# B&R Automation Studio project Soiled_PLC (part 7)

#### 12_sp2Cyclic.ab
```automation-basic
PROGRAM _CYCLIC
	(* cyclic program *)

;---------------------------------------
;Sequence 12 - SP2 Single point 2 D[912]
;---------------------------------------

;Inputs

I_PaddleInPosition		= X[9].X08
I_BagInIncline			= X[9].X07
;I_BagOutAtTop           = X[7].X13

O_OpenBufferStop		= FALSE
O_RunMotor 				= FALSE

I_BagAtOutgoingBuffer	= FALSE
O_OutgoingBufferOpen	= FALSE

Request.IC[1]			= FALSE
Enable.BSF[1]          = FALSE

Alarm[18].Name 			= 0
Alarm[18].Bag			= 10005
Alarm[18].Beacon		= TRUE
Alarm[18].Extra			= 0
Alarm[18].Time			= 3000

;Setup Sequence
STEP = D[918]
;Setup Pulse contact
PLS = (STEP <> LASTSTEP)
LASTSTEP = STEP

;Sequence
;Step 0 - Disabled
IF (STEP = 0) THEN
	;Disabled
ENDIF

;Run Incline until paddle in position
IF (STEP = 1) THEN
	O_RunMotor = NOT I_PaddleInPosition
	IF I_PaddleInPosition THEN
		D[918] = 2
	ENDIF
	IF NOT Std.EStop THEN
		Alarm[18].Name = almSwitchFault
	ENDIF
ENDIF

;request a bag to SP6
IF (STEP = 2) THEN

	IF (Request.BSF[1]  AND NOT Std.HaltSys) THEN
		D[918] = 3
	ENDIF
	;IF (Bag[266].Cat > 0) AND NOT I_BagAtBuffer THEN
		;Alarm[12].Name 	= almBagNotAtProx
		;Alarm[12].Bag	= 266
	;ELSE IF (Bag[266].Cat = 0) AND I_BagAtBuffer THEN
		;Alarm[12].Name 	= almBagNotShownOnScreen
		;Alarm[12].Bag	= 266
	;ENDIF
ENDIF

;Wait for bag to arrive
IF (STEP = 3) THEN
	Enable.BSF[1] 	= TRUE

	IF I_BagInIncline THEN
		D[918] = 4
	ENDIF
	Alarm[18].Name = almBagNotArrived
ENDIF

;Let bag settle at base of incline
TON_10ms((STEP = 4),300,BagSettled,BagSettledET)
IF (STEP = 4) THEN

	IF BagSettled THEN
		D[918] = 5
	ENDIF
ENDIF

;Move Bag up incline
TON_10ms((STEP = 5),500,BagNearTop,BagNearTopET)
TON_10ms(((STEP = 5) AND NOT I_BagInIncline),1000,CloseBufferStop,CloseBufferStopET)
IF (STEP = 5) THEN
	;O_OpenBufferStop 	= NOT CloseBufferStop
	O_RunMotor 			= NOT BagNearTop
	IF BagNearTop  THEN
		D[918] = 6
	ENDIF
	Alarm[18].Name = almSwitchFault
ENDIF

;Check for space at the ongoing buffer
;Run motor for 0.5 seconds
TON_10ms((STEP = 6),50,RunOn,RunOnET)
IF (STEP = 6) THEN
	O_RunMotor 		= NOT RunOn
	IF NOT Std.HaltSys THEN
		Request.IC[1] = TRUE

			IF Enable.IC[1] THEN
				D[918] = 7
			ENDIF

	ENDIF
ENDIF

;Run incline until bag released / arrive at buffer
IF (STEP = 7) THEN
	O_RunMotor 			= TRUE
	;IF PLS THEN
	;	C[13] = 0
	;ENDIF
	IF NOT Enable.IC[1] THEN
		D[918] = 1
	ENDIF
	Alarm[18].Name = almBagNotReleased
ENDIF

;Alarms
TimerAlarm.IN 	= NOT PLS AND (Alarm[18].Name > 0)
TimerAlarm.PT 	= Alarm[18].Time
TimerAlarm FUB TON_10ms()
Alarm[18].On 	= TimerAlarm.Q
Alarm[18].ET 	= TimerAlarm.ET

;Outputs

Y[13].Y04 = O_RunMotor
END_PROGRAM
```

### Program Logical/Sequences/10ms/19_sic_2 (IEC) - * SP2 Empty bags from SDC1/2

#### 12_sp2.var
```iecst
VAR RETAIN
	STEP : UINT;
	PLS : BOOL;
	LASTSTEP : UINT;
END_VAR
VAR
	TimerAlarm : TON_10ms;
	I_BagAtBuffer : BOOL;
	O_OpenBuffer : BOOL;
	SDC2BufferFullET : TIME;
	SDC2BufferFull : BOOL;
	SettledBufferET : TIME;
	SettledBuffer : BOOL;
	O_OpenSP2BufferStop : BOOL;
	O_SelectPoint : BOOL;
	SP2BufferFull : BOOL;
	SP2BufferFullET : UDINT;
	ParingLoopEnabled : BOOL;
	BagInLoopHasDest : BOOL;
	O_OpenSDC1BufferStop : BOOL;
	BagSettledAtBuffer : BOOL;
	BagSettledAtBufferET : UDINT;
	Alternator : USINT;
	I_PaddleInPosition : BOOL;
	I_BagInIncline : BOOL;
	O_OpenBufferStop : BOOL;
	O_RunMotor : BOOL;
	I_BagAtOutgoingBuffer : BOOL;
	O_OutgoingBufferOpen : BOOL;
	BagSettled : BOOL;
	BagSettledET : UDINT;
	BagNearTop : BOOL;
	BagNearTopET : UDINT;
	CloseBufferStop : BOOL;
	CloseBufferStopET : UDINT;
	RunOn : BOOL;
	RunOnET : UDINT;
	I_BagOutAtTop : BOOL;
	BagAtBuffer : BOOL;
	BagAtBufferET : UDINT;
END_VAR
```

#### 12_sp2Cyclic.ab
```automation-basic
PROGRAM _CYCLIC
	(* cyclic program *)

;---------------------------------------
;Sequence 12 - SP2 Single point 2 D[912]
;---------------------------------------

;Inputs

I_BagAtBuffer			= X[9].X09
I_PaddleInPosition		= X[9].X11
I_BagInIncline			= X[9].X10
I_BagOutAtTop           = FALSE ;X[6].X14

O_OpenBufferStop		= FALSE
O_RunMotor 				= FALSE

I_BagAtOutgoingBuffer	= FALSE
O_OutgoingBufferOpen	= FALSE

;Enable.SIC[2]			= FALSE

Alarm[19].Name 			= 0
Alarm[19].Bag			= 10005
Alarm[19].Beacon		= TRUE
Alarm[19].Extra			= 0
Alarm[19].Time			= 3000

;Setup Sequence
STEP = D[919]
;Setup Pulse contact
PLS = (STEP <> LASTSTEP)
LASTSTEP = STEP

;Sequence
;Step 0 - Disabled
IF (STEP = 0) THEN
	;Disabled
ENDIF

;Run Incline until paddle in position
IF (STEP = 1) THEN
	O_RunMotor = NOT I_PaddleInPosition
	IF I_PaddleInPosition THEN
		D[919] = 2
	ENDIF
	IF NOT Std.EStop THEN
		Alarm[19].Name = almSwitchFault
	ENDIF
ENDIF

;Wait for at buffer
TON_10ms(I_BagAtBuffer,300,BagAtBuffer,BagAtBufferET)
IF (STEP = 2) THEN
	IF (BagAtBuffer  AND NOT Std.HaltSys) THEN
		D[919] = 3
	ENDIF
	;IF (Bag[266].Cat > 0) AND NOT I_BagAtBuffer THEN
		;Alarm[12].Name 	= almBagNotAtProx
		;Alarm[12].Bag	= 266
	;ELSE IF (Bag[266].Cat = 0) AND I_BagAtBuffer THEN
		;Alarm[12].Name 	= almBagNotShownOnScreen
		;Alarm[12].Bag	= 266
	;ENDIF
ENDIF

;Open Buffer stop
IF (STEP = 3) THEN
	O_OpenBufferStop 	= TRUE
	;Enable.SIC[1]		= NOT I_BagInIncline
	IF I_BagInIncline THEN
		D[919] = 4
	ENDIF
	Alarm[19].Name = almBagNotArrived
ENDIF

;Let bag settle at base of incline
TON_10ms((STEP = 4),300,BagSettled,BagSettledET)
IF (STEP = 4) THEN
	;O_OpenBufferStop 	= TRUE
	;IF PLS THEN
	;	Bag[265] = Bag[266]
	;	Bag[266] = Bag[0]
	;ENDIF
	IF BagSettled THEN
		D[919] = 5
	ENDIF
ENDIF

;Move Bag up incline
TON_10ms((STEP = 5),500,BagNearTop,BagNearTopET)
TON_10ms(((STEP = 5) AND NOT I_BagInIncline),1000,CloseBufferStop,CloseBufferStopET)
IF (STEP = 5) THEN
	;O_OpenBufferStop 	= NOT CloseBufferStop
	O_RunMotor 			= NOT BagNearTop
	IF BagNearTop THEN
		D[919] = 6
	ENDIF
	Alarm[19].Name = almSwitchFault
ENDIF

;Check for space at the ongoing buffer
;Run motor for 0.5 seconds
TON_10ms((STEP = 6),50,RunOn,RunOnET)
IF (STEP = 6) THEN
	O_RunMotor 		= NOT RunOn
	IF NOT Std.HaltSys THEN
		;IF (Bag[273].Cat = 0) AND NOT I_BagAtOutgoingBuffer AND NOT O_OutgoingBufferOpen THEN
			;IF Line[15].Clear THEN
			IF Line[24].Clear THEN
				D[919] = 7
			;ELSE
			;	Alarm[13].Name = almSwitchFault
			ENDIF
		;ENDIF
	ENDIF
ENDIF

;Run incline until bag released / arrive at buffer
IF (STEP = 7) THEN
	O_RunMotor = TRUE
	IF PLS THEN
		C[24] = 0
	ENDIF
	IF Line[24].Trip THEN
		D[919] = 1
	ENDIF
	Alarm[19].Name = almBagNotReleased
ENDIF

;Alarms
TimerAlarm.IN 	= NOT PLS AND (Alarm[19].Name > 0)
TimerAlarm.PT 	= Alarm[19].Time
TimerAlarm FUB TON_10ms()
Alarm[19].On 	= TimerAlarm.Q
Alarm[19].ET 	= TimerAlarm.ET

;Outputs
Y[9].Y09 = O_OpenBufferStop
Y[13].Y05 = O_RunMotor
END_PROGRAM
```

### Program Logical/Sequences/10ms/8_sl1 (IEC, version 3.00.6) - *Servo Hoist - 3 position

#### sl3.st - Init, cyclic, exit code
```iecst
(********************************************************************
* COPYRIGHT --
********************************************************************
* PROGRAM: sl4.st
* File: sl4.st
* Author: treamsbottom
* Created: March 6 2019
********************************************************************
* Implementation OF PROGRAM Servo Hoist 4 Postion
********************************************************************)
//V2.00.1 First Release
//V2.00.2 FIX - LoadBag wasn;t being set on belt loaded type
//V2.00.3 FIX - 11/08/2019 - Carriage Move alarms were active when the safety zone was off.
//V2.00.4 CHANGE - 11/08/2019 - If the hoist is out of position on loading step- then move to position
//V2.00.5 ADD 12/08/2019 - Add option to stop full bags being bought into service position
//V3.00.1 CHANGE:TR  22/08/2019 - Load Alarms and timer values from config
//V3.00.2 TR 15/09/2019 - Remove EDGEPOS on deviceOut.Bag reference as this doesn;t work with 1_x points as the bag number can change dynamically
//V3.00.3 TR 18/08/2019	- ADD bag check when bag is being loaded.
//V3.00.4 TR 04/10/2019 - FIX: Additional check on Std.MaxCats due to config mode sets to 0 for first scan
//V3.00.5 TR 06/11/2019 - ADD: Alarm when servo hoist is in error.
//V3.00.6 TR 06/11/2019 - FIX: Don;t clear Comm with Comm[0] as unconfiguried tasks can write to Comm[0]
PROGRAM _INIT
//Configuration
mySeq						:= 8;						//Sequence number
MY_VC;						//SET CONSTANT				//Hoist Number Number
myZone 						:= 2;						//Safety Zone
myBag						:= 222;

allowFullBagsInServicePos	:= TRUE;					//Set this to true, if full bags are allowed into service position. Off by default to prevent squashing full bags

//Options
bulkLoaded					:= 0;						//Is the Hoist bulk Loaded.
requestPrgCode				:= 0;						//Request a PRG code from trackview using this d32 register (Start 100 and increase by 20s MAX is 180
CASE Std.PLCStn OF
	0:
		myHoistID				:= 230 + MY_VC;
	1:
		myHoistID				:= 240 + MY_VC;

END_CASE;

//Option to clear the destination when bag arrives,

alarm						ACCESS ADR(Alarm[mySeq]);
bag							ACCESS ADR(Bag[myBag]);
bag_out						ACCESS ADR(Bag[224]);

pHoist 						ACCESS ADR(OpcUa.VC[myHoistID]);
returnStep					ACCESS ADR(D[7970 + MY_VC]);

position_BagOut				:= 1;
position_BagIn				:= 2;
position_Service			:= 3;

i_bagReleased				ACCESS ADR(X[3].X14);
//Outputs
o_safeStopA					ACCESS ADR (Y[0].Y07);
o_safeStopB					ACCESS ADR (Y[0].Y08);
o_guardMoveDown				ACCESS ADR(Hoist_Safety[MY_VC].O_OpenGuard);
o_guardMoveUp				ACCESS ADR(Hoist_Safety[MY_VC].O_CloseGuard);

#if (MY_VC > MAX_HOIST)
	#error 'MAX_HOIST has not been set correctly'
#endif

END_PROGRAM

PROGRAM _CYCLIC

Bag[217].Cat := 1;
Bag[217].Wgt := DINT_TO_UINT(pHoist.Read.Weight/100);
IF (Bag[217].Bid = 0) AND (BidStn > 0) THEN
	Bag[217].Bid := BidStn;
	BidStn := 0;
END_IF;

Request.VC[1]				:= FALSE;

Enable.VC[1]  				:= FALSE;
guardMoveDown				:= FALSE;

//Bit so we can customise the permission to move if required. FOR USE WITH MOVING TOP RAILS
permission_GetBag		:= TRUE;
permission_ReleaseBag	:= TRUE;
permission_Move			:= NOT Std.HaltSysZone[myZone];

pHoist.Write.PermissionToMove := 0;//We have to set permission to move when we want the hoist move.
pHoist.Write.Heartbeat;//This is taken care of in the server task,
pHoist.Write.LoadBag 	:= 0;	//
pHoist.Write.ReceiveBag := 0;	//Cmd to recieve bag
pHoist.Write.ReleaseBag	:= 0;	//Cmd to release bag
pHoist.Write.TargetPosition;	//Set the position of hoist.

autoMode 				:= pHoist.Read.Auto;

IF (myBag = 0) THEN
	alarm.Bag	:= mySeq + 10000;
ELSE
	alarm.Bag	:= myBag;
END_IF;

alarm.Name 		:= 0;
alarm.Beacon	:= TRUE;
alarm.Extra		:= 0;
alarm.Time		:= 3000;

//Setup Sequence
step := D[900 + mySeq];
//Setup Pulse contact
pls := (step <> lastStep);
lastStep := step;

//clear any latched bits
IF pls THEN
	releaseBag := 0;
END_IF;

//Sequence
IF (step = 0) THEN
	//Disabled
END_IF;

//step 1 - move to emptybag in position
IF (step = 1) THEN
	reqPosition := position_BagIn;
	pHoist.Write.PermissionToMove := permission_Move;
	IF (pHoist.Read.PositionNo = reqPosition) AND pHoist.Read.ReadyToReceive THEN
		D[900 + mySeq] := 2;
	END_IF;
	IF autoMode AND permission_Move THEN
		alarm.Name := ALM_CARRIAGE_MOVE_FAULT;
		alarm.Time := 1500;
	END_IF;
END_IF;

//Step 2 - Give permission to recieve bag
IF (step = 2) THEN
	readyToRecieve := ((bag.Cat = 0) AND (pHoist.Read.PositionNo = reqPosition) AND pHoist.Read.ReadyToReceive AND autoMode);
	pHoist.Write.ReceiveBag := 1;
	reqPosition := position_BagIn;
	IF readyToRecieve AND RequestRel.LU[1] THEN // Bag hs been released to empty bag in
		D[900 + mySeq] := 3;
	ELSIF (bag.Cat > 0) THEN
		alarm.Name := ALM_BAG_DATA_ERROR;
	ELSIF (pHoist.Read.PositionNo <> reqPosition) AND autoMode AND permission_Move THEN // Move to position if the buffer hasn;t already been opened.
		pHoist.Write.PermissionToMove := permission_Move;
		alarm.Name := ALM_CARRIAGE_MOVE_FAULT;
		alarm.Time := 1500;
	END_IF;

END_IF;

//Step 3-- Wait for bag to arrive on carriage.
IF (step = 3) THEN
	reqPosition := position_BagIn;
	pHoist.Write.ReceiveBag := 1;
	IF ((bag.Cat = 0) AND (pHoist.Read.PositionNo = reqPosition) AND pHoist.Read.ReadyToReceive AND autoMode AND RequestRel.LU[1]) THEN
		readyToRecieve := 1;
	END_IF;
	Enable.VC[1] := readyToRecieve;
	IF pHoist.Read.ReceiveBag AND (bag.Cat = 0) THEN
		D[900 + mySeq] := 4;
	ELSIF (((pHoist.Read.PositionNo <> reqPosition) OR NOT pHoist.Read.ReadyToReceive ) AND autoMode AND permission_Move) THEN
		alarm.Name := ALM_CARRIAGE_MOVE_FAULT;
		alarm.Time := 1500;
	END_IF;
ELSE
	readyToRecieve := 0;
END_IF;

//step 4 - move to full bag out
IF (step = 4) THEN
	reqPosition := position_BagOut;
	pHoist.Write.PermissionToMove := permission_Move AND permission_ReleaseBag;
	IF (pHoist.Read.PositionNo = reqPosition) AND NOT Enable.PN[1] THEN //We have no feedback for ready to release!! this is checked in the hoist.
		D[900 + mySeq] := step + 1;
	END_IF;
	IF autoMode AND permission_Move  THEN
		alarm.Name := ALM_CARRIAGE_MOVE_FAULT;
		alarm.Time := 1500;
	ELSIF Enable.PN[1] THEN
			alarm.Name := ALM_GENERAL_SEQUENCE;
			alarm.Time := 500;
	END_IF;
	//We should check the hoist status for any alarms??
END_IF;

//step 5 Request Release full bag out
wieghtCheck := (pHoist.Read.Weight < 55000); // hoist sends to 3 decimal places
IF (step = 5) THEN
	okToRelease := Enable.PN[1] AND wieghtCheck AND NOT i_bagReleased;
	reqPosition := position_BagOut;
	requestRelease := (((bag.Cat > 0) OR (myBag = 0) OR Enable.PN[1]) AND (pHoist.Read.PositionNo = reqPosition) AND autoMode AND NOT Std.HaltSysZone[myZone]);
	Request.VC[1]	:= requestRelease;
	IF NOT wieghtCheck THEN
		alarm.Name := almBagOverWeight;
		alarm.Time	:= 500;
	ELSIF requestRelease AND okToRelease  THEN
		D[900 + mySeq] := 6;
	ELSIF (myBag > 0) AND (bag.Cat = 0) THEN
		alarm.Name := ALM_BAG_DATA_ERROR;
		alarm.Time := 0;
	END_IF;
END_IF;

//Step 6 Send the command to release the full bag

bagReleased := (i_bagReleased OR NOT Enable.PN[1]);

IF (step = 6) THEN
	okToRelease :=  Enable.PN[1] AND wieghtCheck;
	reqPosition := position_BagOut;
	IF okToRelease AND (pHoist.Read.PositionNo = reqPosition) AND NOT Std.HaltSysZone[myZone] AND autoMode THEN
		releaseBag := 1;
	END_IF;
	pHoist.Write.ReleaseBag := releaseBag;

	IF NOT wieghtCheck THEN
		alarm.Name := almBagOverWeight;
		alarm.Time	:= 500;
	END_IF;
	IF bagReleased AND releaseBag THEN
//		bag_out := bag;
//		bag := Bag[0];
		D[900 + mySeq] := 1;
	END_IF;
	IF NOT Std.HaltSysZone[myZone] THEN
		alarm.Name := ALM_BAG_NOT_RELEASED;
		alarm.Time := 1500;
	END_IF;
ELSE
	releaseBag := 0;
END_IF;

//Move to service position
IF (step = 90) THEN
	pHoist.Write.PermissionToMove := 1;
	reqPosition := position_Service;
	IF (pHoist.Read.PositionNo = position_Service) THEN //We have no feedback for ready to release!! this is checked in the hoist.
		D[900 + mySeq] := 91;
	END_IF;
	IF autoMode AND permission_Move THEN
		alarm.Name := ALM_CARRIAGE_MOVE_FAULT;
		alarm.Time := 1500;
	END_IF;
END_IF;

//step 91 -- In safe position- Wait for zone to be opened or request to go off
IF (step = 91) THEN
	IF 	SafetyZone[myZone].AccessRequested AND NOT SafetyZone[myZone].Zone_Status THEN
		D[900 + mySeq] := 92;
	ELSIF NOT SafetyZone[myZone].AccessRequested THEN
		D[900 + mySeq] := returnStep;
	ELSIF Hoist_Safety[MY_VC].OutOfPosition THEN
		alarm.Name := ALM_SWITCH_FAULT;
		alarm.Time := 200;
	END_IF;
END_IF;

//step 92 -- Door opened-  wait for safety OK
IF (step = 92) THEN
	IF SafetyZone[myZone].Zone_Status THEN
		D[900 + mySeq] := returnStep;
	END_IF;
END_IF;

IF allowFullBagsInServicePos THEN
	fullBagOnHoist := 0;
ELSE
	fullBagOnHoist := (((bag.Cat > 0) AND (bag.Cat <> Std.MaxCats)) OR ((step > 3) AND (step < 90)));
END_IF;

//Code to request the hoist to move to service position.
IF SafetyZone[myZone].AccessRequested AND (step > 0) AND (step <> 3) AND (step <> 6) AND (step < 90)  AND autoMode AND NOT releaseBag AND NOT fullBagOnHoist THEN
	D[900 + mySeq] := 90;
	CASE step OF
		2:
			returnStep := (step - 1);
		ELSE
			returnStep := step;
	END_CASE;
END_IF;

o_safeStopA	 	:= (step = 3) AND (pHoist.Read.ReadyToReceive OR TestSystem);//Safety stops
o_safeStopB		:= o_safeStopA;

pHoist.Write.BagInTransit := (step = 3) OR releaseBag; //Stop the hoist going into manual mode while a bag is moving.
pHoist.Write.TargetPosition := reqPosition;
o_guardMoveDown := guardMoveDown;
o_guardMoveUp := NOT guardMoveDown;

IF (pHoist.Read.Error OR NOT pHoist.Read.Heartbeat) AND NOT Std.HaltSysZone[myZone] THEN
	alarm.Name := ALM_SERVO_HOIST;
	IF pHoist.Read.Error THEN
		alarm.Time := 400;
	ELSE
		alarm.Time := 3000;
	END_IF;
END_IF;

//Alarms
timerAlarm(IN := NOT pls AND (alarm.Name > 0) AND (alarm.Name = lastAlarm) ,PT:= alarm.Time);
lastAlarm := alarm.Name;

alarm.On 	:= timerAlarm.Q;
alarm.ET 	:= timerAlarm.ET;

END_PROGRAM
```

#### sl3.var - Local variables
```iecst
VAR
	mySeq : UINT;
END_VAR
VAR CONSTANT
	MY_VC : USINT := 1;
END_VAR
VAR
	myZone : USINT;
	myBag : UINT;
	alarm : REFERENCE TO Alm;
	bag : REFERENCE TO Bag_typ;
	bag_out : REFERENCE TO Bag_typ;
	myHoistID : USINT;
	returnStep : REFERENCE TO UINT;
	pHoist : REFERENCE TO OpcUa_VC_type;
	position_BagOut : USINT;
	position_Loading : USINT;
	position_BagIn : USINT;
	position_Service : USINT;
	o_guardMoveUp : REFERENCE TO BOOL;
	o_guardMoveDown : REFERENCE TO BOOL;
	o_safeStopB : REFERENCE TO BOOL;
	o_safeStopA : REFERENCE TO BOOL;
	autoMode : BOOL;
	step : UINT;
	permission_Move : BOOL;
	pls : BOOL;
	lastStep : UINT;
	timerAlarm : TON_10ms;
	reqPosition : USINT;
	readyToRecieve : BOOL;
	okToRelease : BOOL;
	requestRelease : BOOL;
	releaseBag : BOOL;
	f_trig_Released : F_TRIG;
	r_trig_Released : R_TRIG;
	guardMoveDown : BOOL;
	permission_GetBag : BOOL;
	permission_ReleaseBag : BOOL;
	bulkLoaded : BOOL;
	moveGuardDown : BOOL;
	unloadFinished : BOOL;
	myPrg : USINT;
	myCat : UDINT;
	myCus : UDINT;
	myWgt : UINT;
	myMis : UDINT;
	myCnt : UINT;
	myBid : UDINT;
	myDst : UINT;
	myTime : DATE_AND_TIME;
	requestPrgCode : UINT;
	myReportStn : UINT;
	allowFullBagsInServicePos : BOOL; (*Option to allow full bags into service position*)
	fullBagOnHoist : BOOL;
	bagOnCarriage : BOOL;
	lastAlarm : UINT;
	i_bagReleased : REFERENCE TO BOOL;
	bagReleased : BOOL;
	wieghtCheck : BOOL;
END_VAR
```

### Program Logical/Sequences/10ms/10_ebt (IEC) - * EBT Empty bag transfer from SDC2

#### 10_ebt.var
```iecst
VAR RETAIN
	STEP	:UINT;
	PLS	:BOOL;
	LASTSTEP	:UINT;
END_VAR

VAR
	O_OpenBufferStop	:BOOL;
	SettledAtBufferET	:TIME;
	I_BagAtBuffer	:BOOL;
	SettledAtBuffer	:BOOL;
	O_SPI1BufferStopOpen	:BOOL;
	I_BagAtSPI1BufferStop	:BOOL;
	TimerAlarm	:TON_10ms;
	O_SelectPoint	:BOOL;
END_VAR
```

#### 10_ebtCyclic.ab
```automation-basic
PROGRAM _CYCLIC
	(* cyclic program *)

;-----------------------------------------------------
;Sequence 10 - EBT Empty bag transfer from SDC2 D[910]
;-----------------------------------------------------

;Inputs

I_BagAtBuffer			= X[6].X13

O_OpenBufferStop		= FALSE
Enable.DC[1]           = FALSE
O_SelectPoint           = FALSE

I_BagAtSPI1BufferStop	= X[8].X12
O_SPI1BufferStopOpen	= Y[8].Y12

Alarm[10].Name 			= 0
Alarm[10].Bag			= 266
Alarm[10].Beacon		= TRUE
Alarm[10].Extra			= 0
Alarm[10].Time			= 3000

;Setup Sequence
STEP = D[910]
;Setup Pulse contact
PLS = (STEP <> LASTSTEP)
LASTSTEP = STEP

IF (Bag[266].Cat > 0) AND (Bag[266].Bid = 0) AND (BidStn > 0) THEN
	Bag[266].Bid = BidStn
	BidStn = 0
ENDIF

;Sequence
;Step 0 - Disabled
IF (STEP = 0) THEN
	;Disabled
ENDIF

;Step 1 - Wait for space at SPI1 buffer
IF (STEP = 1) THEN
	IF (Line[17].Clear AND NOT I_BagAtSPI1BufferStop AND NOT O_SPI1BufferStopOpen AND NOT Std.HaltSys) THEN
		D[910] = 2
	ENDIF
ENDIF

;Step 2 - Wait for bag at SDC2 empty bag buffer and enable from offgoing
TON_10ms(I_BagAtBuffer,300,SettledAtBuffer,SettledAtBufferET)
IF (STEP = 2) THEN
	IF EnableSDC2Empty THEN
		IF Request.DC[1] THEN
			D[910] = 3
		ELSE IF SettledAtBuffer  THEN
			D[910] = 4
		ENDIF
	ENDIF
ENDIF

;Enable SDC1
IF (STEP = 3) THEN
	Enable.DC[1] = (D[905] <= 2)
	O_SelectPoint = (D[905] <= 2)
	IF PLS THEN
		C[17] = 0
		Bag[266].Prg = Std.MaxProg
		Bag[266].Cat = Std.MaxCats
	ENDIF
	IF Line[17].Trip THEN
		D[910] 		= 1
		Bag[266] 	= Bag[0]
	ENDIF
	Alarm[10].Name = almBagNotArrived
ENDIF

;Step 3 - Transfer empty from SDC2
IF (STEP = 4) THEN
	O_OpenBufferStop = (D[905] <= 2)
	IF PLS THEN
		C[17] = 0
		Bag[266].Prg = Std.MaxProg
		Bag[266].Cat = Std.MaxCats
	ENDIF
	IF Line[17].Trip THEN
		D[910] 		= 1
		Bag[266] 	= Bag[0]
	ENDIF
	Alarm[10].Name = almBagNotArrived
ENDIF

;Alarms
TimerAlarm.IN 	= NOT PLS AND (Alarm[10].Name > 0)
TimerAlarm.PT 	= Alarm[10].Time
TimerAlarm FUB TON_10ms()
Alarm[10].On 	= TimerAlarm.Q
Alarm[10].ET 	= TimerAlarm.ET

;Outputs
Y[6].Y13 = O_OpenBufferStop
Y[8].Y02 = O_SelectPoint
END_PROGRAM
```

### Program Logical/Sequences/10ms/13_spc1 (IEC, version 1.00.0) - * SPC1 Empty bag down

#### 13_spc1Cyclic.ab
```automation-basic
PROGRAM _CYCLIC
	(* cyclic program *)

;----------------------------------------------
;Sequence 13 - SPC1 Pneumatic Conveyor 1 D[913]
;----------------------------------------------

;Inputs
I_CarrAtTop				= X[5].X09
I_CarrAtBottom			= X[5].X10
I_BagOnCarr				= X[5].X11
I_BagReleased			= FALSE ;X[13].X04
I_BagAtBuffer			= X[5].X12

I_BagAtLLBuff			= FALSE ;X[12].X01
O_LLBuffOpen			= FALSE ;Y[12].Y01

O_OpenBuffer			= FALSE
O_MoveCarrUp			= FALSE
O_MoveCarrDown			= FALSE
O_OpenCarrStop			= FALSE

Alarm[13].Name 			= 0
Alarm[13].Bag			= 10013
Alarm[13].Beacon		= FALSE
Alarm[13].Extra			= 0
Alarm[13].Time			= 3000

;Setup Sequence
STEP = D[913]
;Setup Pulse contact
PLS = (STEP <> LASTSTEP)
LASTSTEP = STEP

;Sequence
IF (STEP = 0) THEN
	;Disabled
ENDIF

;Move carriage up to top position
IF (STEP = 1) THEN
	O_MoveCarrUp = TRUE
	IF I_CarrAtTop THEN
		D[913] = 2
	ENDIF
	IF NOT Std.EStop THEN
		Alarm[13].Name = almCarriageMoveFault
	ENDIF
ENDIF

;Check Status
IF (STEP = 2) THEN
	IF (NOT I_BagOnCarr AND NOT I_CarrAtBottom) THEN
		D[913] = 3
	ENDIF
	IF I_BagOnCarr OR I_CarrAtBottom THEN
		Alarm[13].Name = almSwitchFault
	ENDIF
ENDIF

;Wait for bag at buffer
TON_10ms(I_BagAtBuffer,300,SettledBuffer,SettledBufferET)
IF (STEP = 3) THEN
	IF SettledBuffer AND NOT Std.HaltSys THEN
		D[913] = 4
	ENDIF
ENDIF

;Open Buffer stop - Enable
IF (STEP = 4) THEN
	O_OpenBuffer 	= (NOT I_BagOnCarr AND I_CarrAtTop)
	;Enable.SVC[4] 	= (NOT I_BagOnCarr AND I_CarrAtBottom)
	IF I_BagOnCarr THEN
		D[913] = 5
	ENDIF
	Alarm[13].Name = almBagNotArrived
ENDIF

;Let bag settle on carriage
TON_10ms(I_BagOnCarr,300,BagSettledOnCarr,BagSettledOnCarrET)
IF (STEP = 5) THEN
	IF BagSettledOnCarr THEN
		D[913] = 6
	ENDIF
	Alarm[13].Name = almBagNotSettled
ENDIF

;Move Carriage down to bottom position
IF (STEP = 6) THEN
	O_MoveCarrDown = TRUE
	IF I_CarrAtBottom THEN
		D[913] = 7
	ENDIF
	IF NOT Std.EStop THEN
		Alarm[13].Name = almCarriageMoveFault
	ENDIF
ENDIF

;Check if buffer is clear
IF (STEP = 7) THEN
	;IF (Line[33].Clear AND NOT I_BagAtLLBuff AND NOT O_LLBuffOpen AND NOT Std.HaltSysLoading) THEN
	IF Enable.BSN[1] THEN
		D[913] = 8
	ENDIF
	;IF NOT Std.HaltSys THEN
	;	IF I_BagReleased THEN
	;		Alarm[13].Name = almSwitchFault
	;	ENDIF
	;ENDIF
ENDIF

;Open carriage stop let bag into buffer
IF (STEP = 8) THEN
	O_OpenCarrStop = TRUE
	;IF PLS THEN
	;	C[33] = 0
	;ENDIF
	;IF Line[33].Trip THEN
	IF NOT Enable.BSN[1] THEN
		D[913] = 9
	ENDIF
	IF NOT Std.EStop THEN
		Alarm[13].Name = almBagNotReleased
	ENDIF
ENDIF

;Check Top position switch
IF (STEP = 9) THEN
	IF NOT I_CarrAtTop THEN
		D[913] = 1
	ENDIF
	Alarm[13].Name = almSwitchFault
ENDIF

;Alarms
TimerAlarm.IN 	= NOT PLS AND (Alarm[13].Name > 0)
TimerAlarm.PT 	= Alarm[13].Time
TimerAlarm FUB TON_10ms()
Alarm[13].On 	= TimerAlarm.Q
Alarm[13].ET 	= TimerAlarm.ET

;PLC Outputs
;-----------
Y[7].Y16 		= (O_OpenBuffer 	AND I_CarrAtTop)
Y[2].Y03 		= (O_MoveCarrUp 	AND NOT I_CarrAtTop)
Y[2].Y07 		= (O_MoveCarrDown 	AND NOT I_CarrAtBottom)
Y[2].Y12 		= (O_OpenCarrStop 	AND I_CarrAtBottom)

;Don't allow forcing of carriage movement and carriage stop
YForceDisable[7].Y16 = TRUE
YForceDisable[2].Y03 = TRUE
YForceDisable[2].Y07 = TRUE
YForceDisable[2].Y12 = TRUE

END_PROGRAM
```

#### 13_spc1.var
```iecst
VAR RETAIN
	I_CarrAtTop	:BOOL;
	I_CarrAtBottom	:BOOL;
	STEP	:UINT;
	PLS	:BOOL;
	LASTSTEP	:UINT;
	O_MoveCarrUp	:BOOL;
	O_OpenCarrStop	:BOOL;
	O_MoveCarrDown	:BOOL;
	I_BagOnCarr	:BOOL;
END_VAR

VAR
	O_OpenBuffer	:BOOL;
	SettledBuffer	:BOOL;
	SettledBufferET	:TIME;
	I_BagAtBuffer	:BOOL;
	BagSettledOnCarr	:BOOL;
	BagSettledOnCarrET	:TIME;
	I_BagReleased	:BOOL;
	TimerAlarm	:TON_10ms;
	I_BagAtLLBuff	:BOOL;
	O_LLBuffOpen	:BOOL;
END_VAR
```

### Program Logical/Sequences/10ms/16_sdc3 (IEC, version 1.00.0) - * SDC3 Wash-extractors

#### 16_sdc3Cyclic.ab
```automation-basic
PROGRAM _CYCLIC
	(* cyclic program *)

;Sequence 16 - Discharger 3 D[916]

;-----------------------------------------
;Revision 1.00 19/12/2005 D.J. First Issue
;-----------------------------------------

DischargerEnable 		= (NOT Std.HaltSys)

I_BagAtBuffer			= FALSE
I_BagAtDischarger		= X[8].X07
I_OpenBag				= X[8].X08
I_LoadDropped			= X[8].X08
I_BagReleased			= FALSE
I_BagEmpty			  	= TRUE

I_BagAtEmptyBuffer		= FALSE ;X[11].X07
O_EmptyBagBufferOpen	= FALSE ;Y[11].Y07

O_BagReady				= FALSE
O_OpenBuffer 			= FALSE
O_Steadys				= FALSE
O_Closer				= FALSE
O_OpenBag				= FALSE
O_OpenStop				= FALSE

;Enable.DC[1]			= FALSE
Request.DC[3]			= FALSE

;Alarm
Alarm[16].Name 			= almNoAlarm ;Clear sequence alarm name
Alarm[16].Bag 			= 263
Alarm[16].Beacon		= TRUE
Alarm[16].Extra			= 0
Alarm[16].Time			= 3000

;Setup Sequence
STEP = D[916]
;Setup Pulse contact
PLS = (STEP <> LASTSTEP)
LASTSTEP = STEP

;Step 0 - Disabled
IF (STEP = 0) THEN
	;Disabled
ENDIF

;Check Status - Bag settled at buffer, no bag at discharger, bag at buffer on screen and no bag at discharger on the screen
TON_10ms(I_BagAtBuffer,300,SettledAtBuffer,SettledAtBufferET)
IF (STEP = 1) THEN
	;IF (DischargerEnable AND SettledAtBuffer AND NOT I_BagAtDischarger AND (Bag[261].Cat > 0) AND (Bag[263].Cat = 0) AND NOT Std.HaltSys) THEN
	IF (DischargerEnable AND NOT I_BagAtDischarger AND (Bag[263].Cat = 0) AND NOT Std.HaltSys) THEN
		D[916] = 2
	ENDIF
	IF (Bag[263].Cat > 0) THEN
		Alarm[16].Name = almBagDataError
	ELSE IF I_BagAtDischarger THEN
		Alarm[16].Name = almSwitchFault
	;ELSE IF (Bag[263].Cat > 0) AND NOT I_BagAtBuffer THEN
	;	Alarm[16].Name 	= almBagDataError
	;	Alarm[16].Bag	= 263
	;ELSE IF (Bag[261].Cat = 0) AND I_BagAtBuffer THEN
	;	Alarm[16].Name 	= almBagNotShownOnScreen
	;	Alarm[16].Bag	= 261
	ENDIF
ENDIF

;Wait for bag in discharger
IF (STEP = 2) THEN
	;Enable.DC[1]	= TRUE
	;O_OpenBuffer 	= TRUE
	IF I_BagAtDischarger THEN
		D[916] = 3
	ENDIF
	;Alarm[16].Name = almBagNotArrived
ENDIF

;Let bag settle in discharger
TON_10ms(((STEP = 3) AND I_BagAtDischarger),1000,SettledAtDischarger,SettledAtDischargerET)
IF (STEP = 3) THEN
	IF PLS  AND (Bag[263].Cat = 0) AND (Bag[252].Cat > 0) THEN
		Bag[252].Dst = 0
		Bag[263]     = Bag[252]
		Bag[252]     = Bag[0]
	ENDIF
	IF SettledAtDischarger THEN
		D[916] = 4
	ENDIF
	IF (Bag[263].Cat = Std.MaxCats) THEN
		D[916] = 11
	ENDIF
	Alarm[16].Name = almBagNotSettled
ENDIF

;Allow steadys to move down
TON_10ms((STEP = 4),400,SteadysDown,SteadysDownET)
IF (STEP = 4) THEN
	IF (SteadysDown AND NOT I_OpenBag) THEN
		D[916] = 5
	ENDIF
	IF I_OpenBag THEN
		Alarm[16].Name = almSwitchFault
	ENDIF
ENDIF

;Steady cylinders on from steps 4 - 9
O_Steadys = ((STEP >= 4) AND (STEP <= 9))

;Bag opener on from step 5 - 8
O_OpenBag = ((STEP >= 6) AND (STEP <= 8))

;Bag Ready to Washing Machine
IF (STEP = 5) THEN
	O_BagReady = TRUE
	IF I_OpenBag OR TestDischarger THEN
		D[916] = 6
	ENDIF
ENDIF

;Set LoadDropped to False
IF (STEP <> 6) THEN
	LoadDropped = FALSE
ENDIF

;Open Bag Until LoadDropped recieved and has been open for 6 seconds
TON_10ms((STEP = 6),600,MinOpen,MinOpenET) ;ET means Elapsed Time
IF (STEP = 6) THEN

	IF NOT I_OpenBag OR TestDischarger THEN
	;IF I_BagEmpty THEN
		LoadDropped = TRUE
	ENDIF

	IF (LoadDropped AND MinOpen) THEN
		;Write Report
		;------------
		IF (ReportUnloading[3].Cat = 0) THEN
			ReportUnloading[3].Cat = UINT(Bag[263].Cat)	;Category
			ReportUnloading[3].Cus = Bag[263].Cus		;Customer
			ReportUnloading[3].Wgt = Bag[263].Wgt		;Weight
			ReportUnloading[3].Cnt = 0					;Count
			ReportUnloading[3].Stn = 0					;Station
			ReportUnloading[3].Mcn = 3					;Machine
		ENDIF
	ENDIF
	IF (LoadDropped AND MinOpen) THEN
		D[916] = 7
	ENDIF
	Alarm[16].Name = almLoadNotDropped
ENDIF

;Change display to empty bag
IF (STEP = 7) THEN
	O_BagReady = Std.Clock500ms
	IF (I_OpenBag OR TestDrop) THEN
		Bag[263].Prg 	= Std.MaxProg
		Bag[263].Cat 	= Std.MaxCats
		D[916] 			= 8
	ENDIF
	Alarm[16].Name = almGeneralSequence
ENDIF

;Close bag
TON_10ms((STEP = 8),700,CloserDown,CloserDownET)
IF (STEP = 8) THEN
	O_Closer = TRUE
	IF CloserDown THEN
		D[916] = 9
	ENDIF
ENDIF

;Allow closer to go back up
TON_10ms((STEP = 9),700,CloserUp,CloserUpET)
IF (STEP = 9) THEN
	IF CloserUp THEN
		D[916] = 10
	ENDIF
ENDIF

;Allow steadys to go up
TON_10ms((STEP = 10),400,SteadyUp,SteadyUpET)
IF (STEP = 10) THEN
	IF SteadyUp THEN
		D[916] = 11
	ENDIF
ENDIF

;Check for space on empty bag buffer
IF (STEP = 11) THEN
	Request.DC[3] = TRUE
	IF Enable.DC[3] THEN
		D[916] = 12
	ENDIF
ENDIF

;Open buffer stop - unitl bag out
IF (STEP = 12) THEN
	O_OpenStop 	= TRUE
	Bag[263] 	= Bag[0]
	IF NOT Enable.DC[3] THEN
		D[916] = 1
	ENDIF
	Alarm[16].Name = almBagNotReleased
ENDIF

;Alarms
TimerAlarm.IN 	= NOT PLS AND (Alarm[16].Name > 0)
TimerAlarm.PT 	= Alarm[16].Time
TimerAlarm FUB TON_10ms()
Alarm[16].On 	= TimerAlarm.Q
Alarm[16].ET 	= TimerAlarm.ET

;Outputs
Y[8].Y08 	= O_BagReady
;Y[6].Y01 	= O_OpenBuffer
Y[8].Y09 	= O_Steadys
Y[8].Y10 	= O_OpenBag
Y[8].Y05 	= O_Closer
Y[8].Y11 	= O_OpenStop
END_PROGRAM
```

#### 16_sdc3.var
```iecst
VAR RETAIN
	STEP	:UINT;
	PLS	:BOOL;
	LASTSTEP	:UINT;
	SteadyUp	:BOOL;
	CloserUpET	:TIME;
	SteadysDown	:BOOL;
	SteadysDownET	:TIME;
	LoadDropped	:BOOL;
	SteadyUpET	:TIME;
	CloserDownET	:TIME;
	SettledAtDischargerET	:TIME;
	MinOpenET	:TIME;
	SettledAtDischarger	:BOOL;
	CloserDown	:BOOL;
	MinOpen	:BOOL;
	CloserUp	:BOOL;
	SettledAtBuffer	:BOOL;
	SettledAtBufferET	:TIME;
	I_BagAtBuffer	:BOOL;
	O_OpenStop	:BOOL;
	O_OpenBag	:BOOL;
	O_Steadys	:BOOL;
	O_OpenBuffer	:BOOL;
	O_Closer	:BOOL;
	I_BagAtDischarger	:BOOL;
	I_OpenBag	:BOOL;
	I_LoadDropped	:BOOL;
	TestDrop	:BOOL;
END_VAR

VAR
	DischargerEnable	:BOOL;
	TestDischarger	:BOOL;
	I_BagEmpty	:BOOL;
	O_BagReady	:BOOL;
	I_BagReleased	:BOOL;
	O_EmptyBagBufferOpen	:BOOL;
	I_BagAtEmptyBuffer	:BOOL;
	TimerAlarm	:TON_10ms;
	CodeStep	:BOOL;
	BCD_BIN_CAT	:BCD_BIN_OUTPUT;
	BCD_BIN_CUS	:BCD_BIN_OUTPUT;
	BCD_BIN_WGT	:BCD_BIN_OUTPUT;
END_VAR
```

### Program Logical/Sequences/10ms/19_sic2 (IEC) - *incline

#### ic.st
```iecst
(********************************************************************
 * COPYRIGHT --
 ********************************************************************
 * Program: ic
 * File: ic.st
 * Author: treamsbottom
 * Created: July 17, 2015
 ********************************************************************
 * Implementation of program Incline conveyor.
 ********************************************************************)
//V1.00.1 First Release
PROGRAM _INIT
//Configuration
mySeq					:= 19;		//Sequence number
myIO					:= 10; 	//Incline Conveyor IO module number
myIC					:= 2;		//Incline Conveyor Number
useRequest				:= FALSE; 	//Use the Request bit. Only use when working with x_1_point. otherwise use RequestRelease as the i_bagAtBuffer.
myBuffBag				:= 261;		//Ingoing Buffer bag number
myBag					:= 259;		//Incline bag number
myRelLine				:= 32;
myOutBag				:= Line[myRelLine].LastBag;	//Outgoing buffer bag number

myZone 					:= 0;
//Timer Values
bufferSettleTime		:= 300;  	// Time for bag to settle at buffer in.
moveUpInclineTime		:= 8;//>>IN SECONDS<< // Time to move bag up incline after closing stop.//Min of 4 to shut buffer stop....

alarm						ACCESS ADR(Alarm[mySeq]);
bag							ACCESS ADR(Bag[myBag]);
bag_buff					ACCESS ADR(Bag[myBuffBag]);
bag_out						ACCESS ADR(Bag[myOutBag]);
line_release				ACCESS ADR(Line[myRelLine]);
END_PROGRAM

PROGRAM _CYCLIC
//Inputs
i_paddleInPosition		:= X[myIO].X03;
i_bagAtBuffer			:= X[myIO].X01;
i_bagInIncline			:= X[myIO].X02;
i_BagReleased			:= FALSE;//X[myIO].X05;  //<--- Bag release trip- only to be used in special cases. Take when using tracked bags, as the next sequence will need to copy data into a transit position

i_bagAtBufferOut 		:= X[11].X03; // Any Single bag buffer out IO.
i_bufferOutOpen			:= Y[11].Y03;

//End of inputs.

o_openBuffer			:= FALSE;
o_runMotor				:= FALSE;

Request.IC[myIC] 		:= FALSE;
RequestRel.IC[myIC] 	:= FALSE;

IF (myBag = 0) THEN
	alarm.Bag	:= mySeq + 10000;
ELSE
	alarm.Bag	:= myBag;
END_IF;

alarm.Name 		:= 0;
alarm.Beacon		:= TRUE;
alarm.Extra		:= 0;
alarm.Time		:= 3000;

//Setup Sequence
step := D[900 + mySeq];
//Setup Pulse contact
pls := (step <> laststep);
laststep := step;

//Sequence
IF (step = 0) THEN
	//Disabled
END_IF;

//Run Incline until paddle in position
IF (step = 1) THEN
	o_runMotor := NOT i_paddleInPosition;
	IF i_paddleInPosition THEN
		D[900 + mySeq] := 2;
		Count[mySeq] := Count[mySeq] + 1;
	END_IF;
	IF NOT Std.HaltSysZone[myZone] THEN
		alarm.Name := ALM_SWITCH_FAULT;
	END_IF;
END_IF;

//Wait for at buffer
ton_10ms_SettledBuffer(IN:= i_bagAtBuffer, PT:= bufferSettleTime);
IF (step = 2) THEN
	IF NOT i_bagInIncline THEN
		IF useRequest THEN
			D[900 + mySeq] := 3;
		ELSE
			IF ton_10ms_SettledBuffer.Q THEN
				IF (myBuffBag > 0) THEN
					IF (bag_buff.Cat > 0) AND (bag.Cat = 0) THEN
						D[900 + mySeq] := 3;
					ELSIF (bag_buff.Cat = 0) THEN
						alarm.Name := ALM_BAG_DATA_ERROR;
						alarm.Bag := myBuffBag;
					ELSE
						alarm.Name := ALM_BAG_DATA_ERROR;
					END_IF;
				ELSE
					D[900 + mySeq] := 3;
				END_IF;
			ELSIF (myBuffBag > 0) AND (bag_buff.Cat > 0) THEN
				alarm.Name := ALM_BAG_NOT_SETTLED;
			END_IF;
		END_IF;
	ELSE
		alarm.Name := ALM_SWITCH_FAULT;
	END_IF;
END_IF;

//Open Buffer stop
IF (step = 3) THEN
	releaseValid := ((myBag = 0) OR ((bag.Cat = 0) AND (bag_buff.Cat > 0)));
	o_openBuffer	   := releaseValid AND NOT useRequest;
	Request.IC[myIC]  := releaseValid AND useRequest;
	IF i_bagInIncline AND releaseValid THEN
		IF (myBag > 0) THEN
			bag := bag_buff; //Clear empty buffer bag data if used
			bag_buff := Bag[0];
		END_IF;
		D[900 + mySeq] := 4;
	ELSIF (myBag > 0) THEN
		IF (bag.Cat > 0) THEN
			alarm.Name := ALM_BAG_DATA_ERROR;
			alarm.Time := 0;
		ELSIF (bag_buff.Cat = 0) THEN
			alarm.Name := ALM_BAG_DATA_ERROR;
			alarm.Bag := myBuffBag;
			alarm.Time := 0;
		ELSE
			alarm.Name  := ALM_BAG_NOT_ARRIVED;
		END_IF;
	ELSE
		alarm.Name  := ALM_BAG_NOT_ARRIVED;
	END_IF;
END_IF;

ton_10ms_SettledIncline(IN:= (step = 4), PT:= 300);
IF (step = 4) THEN
	o_openBuffer := NOT useRequest;
	IF ton_10ms_SettledIncline.Q THEN
		D[900 + mySeq] := 5;
	END_IF;
END_IF;

//Move Bag up incline
ctu_moveUpIncline(CU:=(step = 5) AND NOT Std.HaltSysZone[myZone] AND Std.Clock1s, RESET := (step <> 5), PV := moveUpInclineTime);
IF (step = 5) THEN
	o_openBuffer 	:= (ctu_moveUpIncline.CV <= 4) AND NOT useRequest;//Close buffer stop after 3 seconds running..
	o_runMotor 		:= TRUE;
	IF ctu_moveUpIncline.Q THEN
		D[900 + mySeq] := 6;
	ELSIF NOT Std.HaltSysZone[myZone] THEN
		alarm.Name := ALM_SWITCH_FAULT;
	END_IF;

END_IF;

//Check for line space.
IF (step = 6) THEN
	releaseValid := (NOT i_bagAtBufferOut AND NOT i_bufferOutOpen AND NOT i_BagReleased AND ((myBag = 0) OR ((bag.Cat > 0) AND (bag_out.Cat = 0))));
	IF (myRelLine > 0) THEN
		IF (line_release.Clear AND releaseValid) THEN
			C[myRelLine] := 0;
			D[900 + mySeq] := 7;
		END_IF;
		IF (line_release.Clear AND i_bagAtBufferOut) THEN
			alarm.Name := ALM_SWITCH_FAULT;
		ELSIF (myBag > 0) AND (bag.Cat = 0) THEN
			alarm.Name := ALM_BAG_DATA_ERROR;
			alarm.Time := 0;
		ELSIF line_release.Clear AND (myOutBag > 0) AND (bag_out.Cat > 0) THEN
			alarm.Name := ALM_BAG_DATA_ERROR;
			alarm.Bag := myOutBag;
			alarm.Time := 0;
		END_IF;
	ELSE
		RequestRel.IC[myIC] := releaseValid;
		IF EnableRel.IC[myIC] AND releaseValid THEN

			D[900 + mySeq] := 7;
		ELSIF (myBag > 0) AND (bag.Cat = 0) THEN
			alarm.Name := ALM_BAG_DATA_ERROR;
			alarm.Time := 0;
		ELSIF (myOutBag > 0) AND (bag_out.Cat > 0) THEN
			alarm.Name := ALM_BAG_DATA_ERROR;
			alarm.Bag := myOutBag;
			alarm.Time := 0;
		END_IF;
	END_IF;
	IF i_BagReleased THEN
		alarm.Name := ALM_SWITCH_FAULT;
		alarm.Time := 0;
	END_IF;
	releaseValid := 0; //Clear this as we are using it as a latch in line 7
END_IF;

//Run motor to release bag.
IF (step = 7) THEN
	IF (NOT i_bagAtBufferOut AND NOT i_bufferOutOpen AND ((myBag = 0) OR ((bag.Cat > 0) AND (bag_out.Cat = 0)))) THEN
		releaseValid := 1;
	END_IF;
	o_runMotor := releaseValid AND NOT Std.HaltSysZone[myZone];
	IF releaseValid THEN
		IF (myBag = 0) THEN
			IF (myRelLine > 0) THEN
				IF line_release.Trip THEN
					D[900 + mySeq] := 1;
				END_IF;
			ELSE
				IF NOT EnableRel.IC[myIC] OR i_BagReleased THEN
					D[900 + mySeq] := 1;
				END_IF;
			END_IF;
			IF NOT Std.HaltSysZone[myZone] THEN
				alarm.Name := ALM_BAG_NOT_RELEASED;
			END_IF;
		ELSE//Use tracking
			IF (myRelLine > 0) THEN
				IF line_release.Trip THEN
					bag_out := bag;
					bag := Bag[0];
					D[900 + mySeq] := 1;
				END_IF;
			ELSE
				IF (i_BagReleased OR NOT EnableRel.IC[myIC]) AND (bag.Cat = 0)  THEN // Make sure data is copied out by enabling sequence.
					D[900 + mySeq] := 1;
				ELSIF NOT EnableRel.IC[myIC] AND (bag.Cat > 0) THEN
					alarm.Name := ALM_BAG_DATA_ERROR;
				END_IF;
			END_IF;
		END_IF;
	ELSIF i_bagAtBufferOut OR i_bufferOutOpen THEN
			alarm.Name := ALM_SWITCH_FAULT;
			alarm.Time := 0;
	ELSIF (myBag > 0) THEN
		IF (bag.Cat = 0) THEN
			alarm.Name := ALM_BAG_DATA_ERROR;
			alarm.Time := 0;
		ELSIF (bag_out.Cat > 0) THEN
			alarm.Name := ALM_BAG_DATA_ERROR;
			alarm.Bag := myOutBag;
			alarm.Time := 0;
		END_IF;
	END_IF;
END_IF;

//-----------------------------------
//PLC Outputs - adjust TO suit system
//-----------------------------------

Y[2].Y14	:= o_runMotor;
Y[myIO].Y01 := o_openBuffer;

//Alarms
timerAlarm(IN := NOT pls AND (alarm.Name > 0),PT:= alarm.Time);

alarm.On 	:= timerAlarm.Q;
alarm.ET 	:= timerAlarm.ET;;

END_PROGRAM
```

### Program Logical/Sequences/10ms/27_sic1 (IEC, version 1.00.5) - *incline

#### ic.st - Implementation code
```iecst
(********************************************************************
 * COPYRIGHT --
 ********************************************************************
 * Program: ic
 * File: ic.st
 * Author: treamsbottom
 * Created: July 17, 2015
 ********************************************************************
 * Implementation of program Incline conveyor.
 ********************************************************************)
//V1.00.1 First Release
PROGRAM _INIT
//Configuration
mySeq					:= 9;		//Sequence number
myIO					:= 6; 	//Incline Conveyor IO module number
myIC					:= 1;		//Incline Conveyor Number
useRequest				:= FALSE; 	//Use the Request bit. Only use when working with x_1_point. otherwise use RequestRelease as the i_bagAtBuffer.
myBuffBag				:= 240;		//Ingoing Buffer bag number
myBag					:= 241;		//Incline bag number
myRelLine				:= 0;
myOutBag				:= Line[myRelLine].LastBag;	//Outgoing buffer bag number

myZone 					:= 0;
//Timer Values
bufferSettleTime		:= 300;  	// Time for bag to settle at buffer in.
moveUpInclineTime		:= 8;//>>IN SECONDS<< // Time to move bag up incline after closing stop.//Min of 4 to shut buffer stop....

alarm						ACCESS ADR(Alarm[mySeq]);
bag							ACCESS ADR(Bag[myBag]);
bag_buff					ACCESS ADR(Bag[myBuffBag]);
bag_out						ACCESS ADR(Bag[myOutBag]);
line_release				ACCESS ADR(Line[myRelLine]);
END_PROGRAM

PROGRAM _CYCLIC
//Inputs
i_paddleInPosition		:= X[myIO].X15;
i_bagAtBuffer			:= X[8].X06;
i_bagInIncline			:= X[myIO].X14;
i_BagReleased			:= FALSE;//X[myIO].X05;  //<--- Bag release trip- only to be used in special cases. Take when using tracked bags, as the next sequence will need to copy data into a transit position

i_bagAtBufferOut 		:= FALSE; // Any Single bag buffer out IO.
i_bufferOutOpen			:= FALSE;

//End of inputs.

o_openBuffer			:= FALSE;
o_runMotor				:= FALSE;

Request.IC[myIC] 		:= FALSE;
RequestRel.IC[myIC] 	:= FALSE;

IF (myBag = 0) THEN
	alarm.Bag	:= mySeq + 10000;
ELSE
	alarm.Bag	:= myBag;
END_IF;

alarm.Name 		:= 0;
alarm.Beacon		:= TRUE;
alarm.Extra		:= 0;
alarm.Time		:= 3000;

//Setup Sequence
step := D[900 + mySeq];
//Setup Pulse contact
pls := (step <> laststep);
laststep := step;

//Sequence
IF (step = 0) THEN
	//Disabled
END_IF;

//Run Incline until paddle in position
IF (step = 1) THEN
	o_runMotor := NOT i_paddleInPosition;
	IF i_paddleInPosition THEN
		D[900 + mySeq] := 2;
		Count[mySeq] := Count[mySeq] + 1;
	END_IF;
	IF NOT Std.HaltSysZone[myZone] THEN
		alarm.Name := ALM_SWITCH_FAULT;
	END_IF;
END_IF;

//Wait for at buffer
ton_10ms_SettledBuffer(IN:= i_bagAtBuffer, PT:= bufferSettleTime);
IF (step = 2) THEN
	IF NOT i_bagInIncline THEN
		IF useRequest THEN
			D[900 + mySeq] := 3;
		ELSE
			IF ton_10ms_SettledBuffer.Q THEN
				IF (myBuffBag > 0) THEN
					IF (bag_buff.Cat > 0) AND (bag.Cat = 0) THEN
						D[900 + mySeq] := 3;
					ELSIF (bag_buff.Cat = 0) THEN
						alarm.Name := ALM_BAG_DATA_ERROR;
						alarm.Bag := myBuffBag;
					ELSE
						alarm.Name := ALM_BAG_DATA_ERROR;
					END_IF;
				ELSE
					D[900 + mySeq] := 3;
				END_IF;
			ELSIF (myBuffBag > 0) AND (bag_buff.Cat > 0) THEN
				alarm.Name := ALM_BAG_NOT_SETTLED;
			END_IF;
		END_IF;
	ELSE
		alarm.Name := ALM_SWITCH_FAULT;
	END_IF;
END_IF;

//Open Buffer stop
IF (step = 3) THEN
	releaseValid := ((myBag = 0) OR ((bag.Cat = 0) AND (bag_buff.Cat > 0)));
	o_openBuffer	   := releaseValid AND NOT useRequest;
	Request.IC[myIC]  := releaseValid AND useRequest;
	IF i_bagInIncline AND releaseValid THEN
		IF (myBag > 0) THEN
			bag := bag_buff; //Clear empty buffer bag data if used
			bag_buff := Bag[0];
		END_IF;
		D[900 + mySeq] := 4;
	ELSIF (myBag > 0) THEN
		IF (bag.Cat > 0) THEN
			alarm.Name := ALM_BAG_DATA_ERROR;
			alarm.Time := 0;
		ELSIF (bag_buff.Cat = 0) THEN
			alarm.Name := ALM_BAG_DATA_ERROR;
			alarm.Bag := myBuffBag;
			alarm.Time := 0;
		ELSE
			alarm.Name  := ALM_BAG_NOT_ARRIVED;
		END_IF;
	ELSE
		alarm.Name  := ALM_BAG_NOT_ARRIVED;
	END_IF;
END_IF;

ton_10ms_SettledIncline(IN:= (step = 4), PT:= 300);
IF (step = 4) THEN
	o_openBuffer := NOT useRequest;
	IF ton_10ms_SettledIncline.Q THEN
		D[900 + mySeq] := 5;
	END_IF;
END_IF;

//Move Bag up incline
ctu_moveUpIncline(CU:=(step = 5) AND NOT Std.HaltSysZone[myZone] AND Std.Clock1s, RESET := (step <> 5), PV := moveUpInclineTime);
IF (step = 5) THEN
	o_openBuffer 	:= (ctu_moveUpIncline.CV <= 4) AND NOT useRequest;//Close buffer stop after 3 seconds running..
	o_runMotor 		:= TRUE;
	IF ctu_moveUpIncline.Q THEN
		D[900 + mySeq] := 6;
	ELSIF NOT Std.HaltSysZone[myZone] THEN
		alarm.Name := ALM_SWITCH_FAULT;
	END_IF;

END_IF;

//Check for line space.
IF (step = 6) THEN
	releaseValid := (NOT i_bagAtBufferOut AND NOT i_bufferOutOpen AND NOT i_BagReleased AND ((myBag = 0) OR ((bag.Cat > 0) AND (bag_out.Cat = 0))));
	IF (myRelLine > 0) THEN
		IF (line_release.Clear AND releaseValid) THEN
			C[myRelLine] := 0;
			D[900 + mySeq] := 7;
		END_IF;
		IF (line_release.Clear AND i_bagAtBufferOut) THEN
			alarm.Name := ALM_SWITCH_FAULT;
		ELSIF (myBag > 0) AND (bag.Cat = 0) THEN
			alarm.Name := ALM_BAG_DATA_ERROR;
			alarm.Time := 0;
		ELSIF line_release.Clear AND (myOutBag > 0) AND (bag_out.Cat > 0) THEN
			alarm.Name := ALM_BAG_DATA_ERROR;
			alarm.Bag := myOutBag;
			alarm.Time := 0;
		END_IF;
	ELSE
		RequestRel.IC[myIC] := releaseValid;
		IF EnableRel.IC[myIC] AND releaseValid THEN

			D[900 + mySeq] := 7;
		ELSIF (myBag > 0) AND (bag.Cat = 0) THEN
			alarm.Name := ALM_BAG_DATA_ERROR;
			alarm.Time := 0;
		ELSIF (myOutBag > 0) AND (bag_out.Cat > 0) THEN
			alarm.Name := ALM_BAG_DATA_ERROR;
			alarm.Bag := myOutBag;
			alarm.Time := 0;
		END_IF;
	END_IF;
	IF i_BagReleased THEN
		alarm.Name := ALM_SWITCH_FAULT;
		alarm.Time := 0;
	END_IF;
	releaseValid := 0; //Clear this as we are using it as a latch in line 7
END_IF;

//Run motor to release bag.
IF (step = 7) THEN
	IF (NOT i_bagAtBufferOut AND NOT i_bufferOutOpen AND ((myBag = 0) OR ((bag.Cat > 0) AND (bag_out.Cat = 0)))) THEN
		releaseValid := 1;
	END_IF;
	o_runMotor := releaseValid AND NOT Std.HaltSysZone[myZone];
	IF releaseValid THEN
		IF (myBag = 0) THEN
			IF (myRelLine > 0) THEN
				IF line_release.Trip THEN
					D[900 + mySeq] := 1;
				END_IF;
			ELSE
				IF NOT EnableRel.IC[myIC] OR i_BagReleased THEN
					D[900 + mySeq] := 1;
				END_IF;
			END_IF;
			IF NOT Std.HaltSysZone[myZone] THEN
				alarm.Name := ALM_BAG_NOT_RELEASED;
				alarm.Time := 6000;
			END_IF;
		ELSE//Use tracking
			IF (myRelLine > 0) THEN
				IF line_release.Trip THEN
					bag_out := bag;
					bag := Bag[0];
					D[900 + mySeq] := 1;
				END_IF;
			ELSE
				IF (i_BagReleased OR NOT EnableRel.IC[myIC]) AND (bag.Cat = 0)  THEN // Make sure data is copied out by enabling sequence.
					D[900 + mySeq] := 1;
				ELSIF NOT EnableRel.IC[myIC] AND (bag.Cat > 0) THEN
					alarm.Name := ALM_BAG_DATA_ERROR;
				END_IF;
			END_IF;
		END_IF;
	ELSIF i_bagAtBufferOut OR i_bufferOutOpen THEN
			alarm.Name := ALM_SWITCH_FAULT;
			alarm.Time := 0;
	ELSIF (myBag > 0) THEN
		IF (bag.Cat = 0) THEN
			alarm.Name := ALM_BAG_DATA_ERROR;
			alarm.Time := 0;
		ELSIF (bag_out.Cat > 0) THEN
			alarm.Name := ALM_BAG_DATA_ERROR;
			alarm.Bag := myOutBag;
			alarm.Time := 0;
		END_IF;
	END_IF;
END_IF;

//-----------------------------------
//PLC Outputs - adjust TO suit system
//-----------------------------------

Y[2].Y09	:= o_runMotor;
Y[8].Y06	:= o_openBuffer;

//Alarms
timerAlarm(IN := NOT pls AND (alarm.Name > 0),PT:= alarm.Time);

alarm.On 	:= timerAlarm.Q;
alarm.ET 	:= timerAlarm.ET;;

END_PROGRAM
```

### Program Logical/Sequences/10ms/21_sbsn_1 (IEC) - * SP2 Empty bags from SDC1/2

#### 12_sp2.var
```iecst
VAR RETAIN
	STEP : UINT;
	PLS : BOOL;
	LASTSTEP : UINT;
END_VAR
VAR
	TimerAlarm : TON_10ms;
	I_BagAtBuffer : BOOL;
	O_OpenBuffer : BOOL;
	SDC2BufferFullET : TIME;
	SDC2BufferFull : BOOL;
	SettledBufferET : TIME;
	SettledBuffer : BOOL;
	O_OpenSP2BufferStop : BOOL;
	O_SelectPoint : BOOL;
	SP2BufferFull : BOOL;
	SP2BufferFullET : UDINT;
	ParingLoopEnabled : BOOL;
	BagInLoopHasDest : BOOL;
	O_OpenSDC1BufferStop : BOOL;
	BagSettledAtBuffer : BOOL;
	BagSettledAtBufferET : UDINT;
	Alternator : USINT;
	I_PaddleInPosition : BOOL;
	I_BagInIncline : BOOL;
	O_OpenBufferStop : BOOL;
	O_RunMotor : BOOL;
	I_BagAtOutgoingBuffer : BOOL;
	O_OutgoingBufferOpen : BOOL;
	BagSettled : BOOL;
	BagSettledET : UDINT;
	BagNearTop : BOOL;
	BagNearTopET : UDINT;
	CloseBufferStop : BOOL;
	CloseBufferStopET : UDINT;
	RunOn : BOOL;
	RunOnET : UDINT;
	I_BagOutAtTop : BOOL;
	BagAtBuffer : BOOL;
	BagAtBufferET : UDINT;
	I_BagStackerNearFull : BOOL;
	BagStackerHasSpace : BOOL;
	BagStackerHasSpaceET : UDINT;
	SIC3BufferFull : BOOL;
	SIC3BufferFullET : UDINT;
	I_OnLineA : BOOL;
	I_TiltA : BOOL;
	I_TiltB : BOOL;
	I_Bagout : BOOL;
	O_SelectLineA : BOOL;
	O_SelectLineB : BOOL;
	O_OpenStops : BOOL;
	O_TiltCylinder : BOOL;
	O_OperatePusher : BOOL;
	PointReset : BOOL;
	PointResetET : UDINT;
	BagAtTilt : BOOL;
	BagAtTiltET : UDINT;
	TiltDown : BOOL;
	TiltDownET : UDINT;
	TiltUp : BOOL;
	TiltUpET : UDINT;
	NotFull : BOOL;
	NotFullET : UDINT;
	Pushed : BOOL;
	SBSN1 : BOOL;
	SBSN1ET : UDINT;
	RequirePusherET : UDINT;
	PushedET : UDINT;
	Pusher : BOOL;
	PusherET : UDINT;
	O_Pusher : BOOL;
END_VAR
```

#### 12_sp2Cyclic.ab
```automation-basic
PROGRAM _CYCLIC
	(* cyclic program *)

;---------------------------------------
;Sequence 12 - SP2 Single point 2 D[912]
;---------------------------------------

;Inputs

I_OnLineA		  		= X[7].X01
I_TiltA					= X[7].X02
I_TiltB					= X[7].X03
I_Bagout				= X[7].X04

O_OpenBufferStop		= FALSE
O_SelectLineA			= FALSE
O_SelectLineB			= FALSE
O_OpenStops				= FALSE
O_TiltCylinder			= FALSE
O_OperatePusher			= FALSE
O_Pusher                = FALSE

Request.BSN[1]			= FALSE
Enable.SP[5]            = FALSE

Alarm[21].Name 			= 0
Alarm[21].Bag			= 10010
Alarm[21].Beacon		= TRUE
Alarm[21].Extra			= 0
Alarm[21].Time			= 3000

;Setup Sequence
STEP = D[921]
;Setup Pulse contact
PLS = (STEP <> LASTSTEP)
LASTSTEP = STEP

;Sequence
IF (STEP = 0) THEN
	;Disabled
ENDIF

;Select Line 'A'
TON_10ms((STEP = 1),100,PointReset,PointResetET)
IF (STEP = 1) THEN
	O_SelectLineA = NOT PointReset
	IF PointReset AND NOT Std.HaltSys THEN
		D[921] = 2
	ENDIF
ENDIF

;give request to SP5
IF ((STEP = 2) OR (STEP = 3)) THEN
	Request.BSN[1] = TRUE
ENDIF

;give request to SP5
;TON_10ms(I_BagAtBuffer,300,BagAtBuffer,BagAtBufferET)
IF (STEP = 2) THEN

	IF Enable.BSN[1] THEN
		D[921] = 3
	ENDIF
ENDIF

;Open buffer stop
IF (STEP = 3) THEN
	O_SelectLineA 		= TRUE
	;O_OpenBufferStop 	= TRUE
	;Enable.SP[5]		= NOT I_OnLineA
	IF I_OnLineA THEN
		D[921] = 4
	ENDIF
	Alarm[21].Name = almBagNotArrived
ENDIF

;Select Line 'B' and Wait for bag in Tilt position
TON_10ms((I_TiltA AND I_TiltB),300,BagAtTilt,BagAtTiltET)
IF (STEP = 4) THEN
	O_SelectLineB = TRUE
	IF BagAtTilt THEN
		D[921] = 5
	ENDIF
	Alarm[21].Name = almBagNotSettled
ENDIF

;Tilt down
TON_10ms((STEP = 5),500,TiltDown,TiltDownET)
TON_10ms(TiltDown,300,Pusher,PusherET)
IF (STEP = 5) THEN
	O_TiltCylinder = TRUE
	O_Pusher       = TiltDown
	IF Pusher THEN
		D[921] = 6
	ENDIF
ENDIF

;Tilt up
TON_10ms((STEP = 6),500,TiltUp,TiltUpET)
IF (STEP = 6) THEN
	IF TiltUp THEN
		D[921] = 7
	ENDIF
	Alarm[21].Time			= 1000
	Alarm[21].Name = almDestinationNotValid
ENDIF

;Check not full
TON_10ms(NOT I_Bagout,300,NotFull,NotFullET)
IF (STEP = 7) THEN
	IF NotFull THEN
		D[921] = 8
	ENDIF
	Alarm[21].Name = almBagNotReleased
ENDIF

;Open stops to release bag
IF (STEP = 8) THEN
	O_OpenStops = TRUE
	IF I_Bagout THEN
		D[921] = 1
	ENDIF
	Alarm[21].Name = almBagNotReleased
ENDIF

;Pusher Cylinder
TON_10ms(I_Bagout AND NOT Pushed,200,SBSN1,SBSN1ET)
TON_10ms((STEP = 8)  AND NOT Pushed,500,O_OperatePusher,RequirePusherET)
TON_10ms(O_OperatePusher,500,Pushed,PushedET)

;ton_10ms_o_operatePusher(IN:= (step = 8) AND NOT ton_10ms_Pushed.Q, PT:= 500);
;ton_10ms_Pushed(IN:= o_operatePusher, PT:= 500);

;Alarms
TimerAlarm.IN 	= NOT PLS AND (Alarm[21].Name > 0)
TimerAlarm.PT 	= Alarm[21].Time
TimerAlarm FUB TON_10ms()
Alarm[21].On 	= TimerAlarm.Q
Alarm[21].ET 	= TimerAlarm.ET

;Outputs
;Y[7].Y01 = O_OpenBufferStop
Y[7].Y01 = O_SelectLineA
Y[7].Y02 = O_SelectLineB
Y[7].Y04 = O_TiltCylinder
Y[7].Y05 = O_OpenStops
Y[7].Y03 = O_OperatePusher
Y[7].Y14 = O_Pusher
END_PROGRAM
```

### Program Logical/Sequences/10ms/22_sbsf_1 (IEC) - * SP2 Empty bags from SDC1/2

#### 12_sp2.var
```iecst
VAR RETAIN
	STEP : UINT;
	PLS : BOOL;
	LASTSTEP : UINT;
END_VAR
VAR
	TimerAlarm : TON_10ms;
	I_BagAtBuffer : BOOL;
	O_OpenBuffer : BOOL;
	SDC2BufferFullET : TIME;
	SDC2BufferFull : BOOL;
	SettledBufferET : TIME;
	SettledBuffer : BOOL;
	O_OpenSP2BufferStop : BOOL;
	O_SelectPoint : BOOL;
	SP2BufferFull : BOOL;
	SP2BufferFullET : UDINT;
	ParingLoopEnabled : BOOL;
	BagInLoopHasDest : BOOL;
	O_OpenSDC1BufferStop : BOOL;
	BagSettledAtBuffer : BOOL;
	BagSettledAtBufferET : UDINT;
	Alternator : USINT;
	I_PaddleInPosition : BOOL;
	I_BagInIncline : BOOL;
	O_OpenBufferStop : BOOL;
	O_RunMotor : BOOL;
	I_BagAtOutgoingBuffer : BOOL;
	O_OutgoingBufferOpen : BOOL;
	BagSettled : BOOL;
	BagSettledET : UDINT;
	BagNearTop : BOOL;
	BagNearTopET : UDINT;
	CloseBufferStop : BOOL;
	CloseBufferStopET : UDINT;
	RunOn : BOOL;
	RunOnET : UDINT;
	I_BagOutAtTop : BOOL;
	BagAtBuffer : BOOL;
	BagAtBufferET : UDINT;
	I_BagStackerNearFull : BOOL;
	BagStackerHasSpace : BOOL;
	BagStackerHasSpaceET : UDINT;
	SIC3BufferFull : BOOL;
	SIC3BufferFullET : UDINT;
	I_OnLineA : BOOL;
	I_TiltA : BOOL;
	I_TiltB : BOOL;
	I_Bagout : BOOL;
	O_SelectLineA : BOOL;
	O_SelectLineB : BOOL;
	O_OpenStops : BOOL;
	O_TiltCylinder : BOOL;
	O_OperatePusher : BOOL;
	PointReset : BOOL;
	PointResetET : UDINT;
	BagAtTilt : BOOL;
	BagAtTiltET : UDINT;
	TiltDown : BOOL;
	TiltDownET : UDINT;
	TiltUp : BOOL;
	TiltUpET : UDINT;
	NotFull : BOOL;
	NotFullET : UDINT;
	Pushed : BOOL;
	SBSN1 : BOOL;
	SBSN1ET : UDINT;
	RequirePusherET : UDINT;
	PushedET : UDINT;
	I_RockSepA : BOOL;
	I_RockSepB : BOOL;
	I_OutLineA : BOOL;
	I_OutLineB : BOOL;
	O_OpenRockSep : BOOL;
	O_LevelCylinder : BOOL;
	O_OpenLineAStop : BOOL;
	O_OpenLineBStop : BOOL;
	LevelClear : BOOL;
	LevelClearET : UDINT;
	SettledInSeps : BOOL;
	SettledInSepsET : UDINT;
	SettledLevel : BOOL;
	SettledLevelET : UDINT;
	LevellerDown : BOOL;
	LevellerDownET : UDINT;
	LevellerUp : BOOL;
	LevellerUpET : UDINT;
	O_LevelCylinderUP : BOOL;
	PRLineClearET : ARRAY[0..5] OF UDINT;
END_VAR
```

#### 12_sp2Cyclic.ab
```automation-basic
PROGRAM _CYCLIC
	(* cyclic program *)

;---------------------------------------
;Sequence 12 - SP2 Single point 2 D[912]
;---------------------------------------

;Inputs
I_RockSepA				= X[7].X07
I_RockSepB				= X[7].X08
I_TiltA					= X[7].X09
I_TiltB					= X[7].X10
I_OutLineA				= X[7].X06
I_OutLineB				= X[7].X11

O_OpenRockSep			= FALSE
O_LevelCylinder			= FALSE
O_OpenLineAStop			= FALSE
O_OpenLineBStop			= FALSE
O_SelectLineA			= FALSE
O_SelectLineB			= FALSE

Request.BSF[1]         = FALSE

Alarm[22].Name 			= 0
Alarm[22].Bag			= 10011
Alarm[22].Beacon		= TRUE
Alarm[22].Extra			= 0
Alarm[22].Time			= 3000

;Setup Sequecne
STEP = D[922]
;Setup Pulse contact
PLS = (STEP <> LASTSTEP)
LASTSTEP = STEP

;Sequence

;Select Line 'A'
TON_10ms((NOT I_TiltA AND NOT I_TiltB),100,LevelClear,LevelClearET)
IF (STEP = 1) THEN
	IF LevelClear AND NOT Std.HaltSys THEN
		D[922] = 2
	ENDIF
	Alarm[22].Name = almSwitchFault
ENDIF

;Open seperators wait for leveller to be ready
TON_10ms(((STEP = 2) AND I_RockSepA AND I_RockSepB),200,SettledInSeps,SettledInSepsET)
IF (STEP = 2) THEN
	O_OpenRockSep = TRUE
	IF SettledInSeps THEN
		D[922] = 3
	ENDIF
	;Alarm[22].Name = almBagNotArrived
ENDIF

;Wait for bag to settle in leveller position
TON_10ms((I_TiltA AND I_TiltB),300,SettledLevel,SettledLevelET)
IF (STEP = 3) THEN
	IF SettledLevel THEN
		D[922] = 4
	ENDIF
	Alarm[22].Name = almBagNotSettled
ENDIF

;Move bag leveller down
TON_10ms((STEP = 4),500,LevellerDown,LevellerDownET)
IF (STEP = 4) THEN
	O_LevelCylinder = TRUE
	IF LevellerDown THEN
		D[922] = 5
	ENDIF
ENDIF

;Allow bag leveller to retract
TON_10ms((STEP = 5),500,LevellerUp,LevellerUpET)
IF (STEP = 5) THEN
	O_LevelCylinderUP = TRUE
	IF LevellerUp THEN
		D[922] = 6
	ENDIF
ENDIF

;Check room in Buffer
IF (STEP = 6) THEN
	IF NOT Std.HaltSys THEN
		Request.BSF[1] = TRUE
		IF Enable.BSF[1] THEN
			D[922] = 7
		ENDIF
	ENDIF
ENDIF

O_SelectLineA = ((STEP <> 8) AND (STEP <> 9))

;Open stop on line 'A'
IF (STEP = 7) THEN
	O_OpenLineAStop = TRUE
	;IF PLS THEN
	;	C[17] = 0
	;ENDIF
	IF I_OutLineA THEN
		D[922] = 8
	ENDIF
	Alarm[22].Name = almBagNotReleased
ENDIF

;Open stop on line 'B'
IF (STEP = 8) THEN
	O_OpenLineBStop = TRUE
	IF I_OutLineB THEN
		D[922] = 9
	ENDIF
	Alarm[22].Name = almBagNotReleased
ENDIF

;Select bag stop and wait for bag out of leveller
IF (STEP = 9) THEN
	O_SelectLineB = TRUE
	IF NOT Enable.BSF[1] THEN
		D[922] = 1
	ENDIF
	Alarm[22].Name = almBagNotReleased
ENDIF

;Alarms
TimerAlarm.IN 	= NOT PLS AND (Alarm[22].Name > 0)
TimerAlarm.PT 	= Alarm[22].Time
TimerAlarm FUB TON_10ms()
Alarm[22].On 	= TimerAlarm.Q
Alarm[22].ET 	= TimerAlarm.ET

;Outputs
Y[7].Y08 = O_OpenRockSep
Y[7].Y11 = O_LevelCylinder
Y[7].Y09 = O_OpenLineAStop
Y[7].Y10 = O_OpenLineBStop
Y[7].Y07 = O_SelectLineA
Y[7].Y06 = O_SelectLineB

;SBS Offgoing Bagstacker Pressure relief
TON_10ms((NOT X[7].X12 AND NOT X[7].X13),500,Y[7].Y12,PRLineClearET[0])

;SPR1-3
TON_10ms((NOT X[4].X13 AND NOT X[4].X14),500,Y[4].Y13,PRLineClearET[1])
TON_10ms((NOT X[5].X13 AND NOT X[5].X14),500,Y[5].Y13,PRLineClearET[2])
TON_10ms((NOT X[4].X13 AND NOT X[7].X14),500,Y[7].Y14,PRLineClearET[3])
TON_10ms((NOT X[7].X15 AND NOT X[7].X16),500,Y[7].Y15,PRLineClearET[4])
END_PROGRAM
```

### Program Logical/Sequences/10ms/24_slu_2 (IEC) - * Loading unit SLU1

#### 3_slu_1.var
```iecst
VAR RETAIN
	STEP : UINT;
	PLS : BOOL;
	LASTSTEP : UINT;
	EBagSettled : BOOL;
	EBagSettledET : TIME;
	O_OpenStop : BOOL;
	O_SteadyCylinders : BOOL;
	LoadingUnitClear : BOOL;
	LoadingUnitClearET : TIME;
END_VAR
VAR
	CompressCount : UINT;
	O_MoveCompressorUp : BOOL;
	SteadysUpET : TIME;
	SteadysUp : BOOL;
	SteadysDown : BOOL;
	SteadysDownET : TIME;
	I_BagAtBuffer : BOOL;
	O_OpenBufferStop : BOOL;
	I_BagInLoadingUnit : BOOL;
	I_BagFrontPast : BOOL;
	SwitchFault : BOOL;
	TimerAlarm : TON_10ms;
	I_CompressorAtTop : BOOL;
	I_CompressorAtBot : BOOL;
	I_CompressorAtMid : BOOL;
	O_MoveCompressorDn : BOOL;
	BagSettledBuffer : BOOL;
	BagSettledBufferET : TIME;
	I_BagAtSVC1Buffer : BOOL;
	O_SVC1BufferOpen : BOOL;
	I_ChuteBlocked : BOOL;
	CompressorDn : BOOL;
	CompressorDnET : UDINT;
	O_MoveDownTop : BOOL;
	O_MoveDownBottom : BOOL;
	CompressorUp : BOOL;
	CompressorUpET : UDINT;
	O_ElephantsFoot : BOOL;
	HaltDownStairs : BOOL;
	I_BagAtSIC1Buffer : BOOL;
	O_SIC1BufferOpen : BOOL;
	BagDropped : BOOL;
	ChuteClear : BOOL;
	ChuteClearET : UDINT;
END_VAR
```

#### 3_slu_1Cyclic.ab
```automation-basic
PROGRAM _CYCLIC
	(* cyclic program *)

;--------------------------------
;Sequence 3 - Loading Unit D[903]
;--------------------------------

;Inputs / Ouputs

I_BagAtBuffer			= X[11].X11
I_BagFrontPast			= X[8].X12
I_BagInLoadingUnit		= X[8].X11

I_ChuteBlocked			= X[8].X16
HaltDownStairs          = NOT X[6].X12

;O_MoveCompressorUp		= FALSE
Request.LU[2]  		= FALSE

I_BagAtSIC1Buffer		= X[11].X15 ;X[12].X11
O_SIC1BufferOpen		= Y[11].Y15 ;Y[12].Y11

O_OpenBufferStop		= FALSE
O_SteadyCylinders		= FALSE
O_OpenStop	 			= FALSE

Enable.SDP[1]			= FALSE

Alarm[24].Name 			= 0
Alarm[24].Bag			= 287
Alarm[24].Beacon		= TRUE
Alarm[24].Extra			= 0
Alarm[24].Time			= 3000

;Setup Sequence
;--------------
STEP = D[924]
;Setup Pulse contact
PLS = (STEP <> LASTSTEP)
LASTSTEP = STEP

IF (STEP = 0) THEN
	;Disabled
ENDIF

;Wait for Empty bag at buffer
SwitchFault = (I_BagFrontPast OR I_BagInLoadingUnit)
TON_10ms(NOT SwitchFault,200,LoadingUnitClear,LoadingUnitClearET)
TON_10ms(I_BagAtBuffer,300,BagSettledBuffer,BagSettledBufferET)
IF (STEP = 1) THEN
	IF BagSettledBuffer AND LoadingUnitClear AND NOT HaltDownStairs THEN
	;IF LoadingUnitClear AND NOT Std.HaltSys THEN
		D[924] = 2
	ENDIF
	IF SwitchFault THEN
		Alarm[24].Name = almSwitchFault
	ENDIF
ENDIF

;Open stops let bag in Loading Unit
IF (STEP = 2) THEN
	O_OpenStop 			= TRUE
	O_OpenBufferStop 	= TRUE
	;Enable.SLU[1]		= NOT I_BagFrontPast
	IF I_BagFrontPast THEN
		D[924] = 3
	ENDIF
	Alarm[24].Name = almBagNotArrived
ENDIF

;Wait for bag to settle
TON_10ms(I_BagInLoadingUnit,700,EBagSettled,EBagSettledET)
IF (STEP = 3) THEN
	IF EBagSettled THEN
		D[924] = 4
	ENDIF
	Alarm[23].Name = almBagNotSettled
ENDIF

;Steady cylinders on from steps 4 - 5
O_SteadyCylinders = ((STEP >= 4) AND (STEP <= 8))

;Move Steady Cylinders down
TON_10ms((STEP = 4),300,SteadysDown,SteadysDownET)
IF (STEP = 4) THEN
	IF (SteadysDown AND (Bag[287].Cat = 0)) THEN
		D[924] = 5
	ENDIF
	IF (Bag[287].Cat <> 0) THEN
		Alarm[4].Name = almBagDataError
	ELSE
		Alarm[4].Name = almNoAlarm
	ENDIF
ENDIF

IF ((NOT STEP = 6) AND (NOT STEP = 8)) THEN
	BagDropped = FALSE
ENDIF

;Wait for request from spd 1
IF (STEP = 5) THEN

	IF Request.SDP[1] THEN
		D[924] = 6
	ENDIF
ENDIF

IF (NOT (STEP = 6) AND NOT (STEP = 8)) THEN
	BagDropped = FALSE
ENDIF

;Wait for linen to pass photo cell
TON_10ms(NOT I_ChuteBlocked,300,ChuteClear,ChuteClearET)
IF (STEP = 6) THEN
	Enable.SDP[1] = TRUE
	Request.LU[2] = TRUE

	IF I_ChuteBlocked THEN
		BagDropped = TRUE
	ENDIF
	IF BagDropped AND ChuteClear and (Bag[287].Cat > 0)and (Bag[287].Wgt < 649)THEN
		D[924] = 9
	ELSE IF BagDropped AND ChuteClear and (Bag[287].Cat > 0)and (Bag[287].Wgt > 649)THEN
		D[924] = 9
	ENDIF

ENDIF

;Wait for request from SDP1
IF (STEP = 7) THEN
	IF (Request.SDP[1] AND (Bag[285].Cat = Bag[287].Cat) AND (Bag[287].Wgt < 650)) THEN
		IF Request.SDP[1] THEN
			D[924] = 8
		ENDIF
	ELSE IF (Request.SDP[1] AND (Bag[285].Cat <> Bag[287].Cat)) THEN
		D[924] = 9
	ELSE IF (Bag[287].Wgt > 650)THEN
		D[924] = 9
	ENDIF
ENDIF

;Wait for linen to pass photo cell
TON_10ms((STEP = 6),300,SteadysUp,SteadysUpET)
IF (STEP = 8) THEN
	Enable.SDP[1] = TRUE
	Request.LU[2] = TRUE
	IF I_ChuteBlocked THEN
		BagDropped = TRUE
	ENDIF
	IF BagDropped AND ChuteClear THEN
		D[924] = 9
	ENDIF
ENDIF

;Allow Steady Cylinders to move up
TON_10ms((STEP = 9),300,SteadysUp,SteadysUpET)
IF (STEP = 9) THEN
	IF SteadysUp THEN
		D[924] = 10
	ENDIF
ENDIF

;Move compressor down
IF (STEP = 10) THEN
	D[924] = 11
ENDIF

;Move compressor up
IF (STEP = 11) THEN
	D[924] = 12
ENDIF

;Check for space at Buffer
IF (STEP = 12) THEN
	IF NOT HaltDownStairs THEN
		IF (Bag[284].Cat = 0) AND NOT I_BagAtSIC1Buffer AND NOT O_SIC1BufferOpen THEN
			IF Line[33].Clear THEN
				C[33]   = 0
				D[924] 	= 13
			ELSE
				;Alarm[3].Name = almSwitchFault
			ENDIF
		ENDIF
	ENDIF
ENDIF

;Open stop - Unitl bag out
IF (STEP = 13) THEN
	O_OpenStop = TRUE
	;IF PLS THEN
	;	C[16] = 0
	;ENDIF
	;IF Line[16].Trip THEN
	IF (C[33]>=1) THEN
		IF ((Bag[287].Cat > 0) AND (Bag[284].Cat = 0)) THEN
			Bag[284] = Bag[287]
			Bag[287] = Bag[0]
		ENDIF
		IF (C[33] >= 1) THEN
			D[924] = 1
		ENDIF
	ENDIF
	Alarm[24].Name = almBagNotReleased
ENDIF

;Alarms
TimerAlarm.IN = NOT PLS AND (Alarm[24].Name > 0)
TimerAlarm.PT = Alarm[24].Time
TimerAlarm FUB TON_10ms()
Alarm[24].On = TimerAlarm.Q
Alarm[24].ET = TimerAlarm.ET

;Outputs
;-------

Y[11].Y11 = O_OpenBufferStop
Y[8].Y12 = O_SteadyCylinders
Y[8].Y11 = O_OpenStop

END_PROGRAM
```

### Program Logical/Sequences/10ms/25_sic_4 (IEC) - * SP2 Empty bags from SDC1/2

#### 12_sp2.var
```iecst
VAR RETAIN
	STEP : UINT;
	PLS : BOOL;
	LASTSTEP : UINT;
END_VAR
VAR
	TimerAlarm : TON_10ms;
	I_BagAtBuffer : BOOL;
	O_OpenBuffer : BOOL;
	SDC2BufferFullET : TIME;
	SDC2BufferFull : BOOL;
	SettledBufferET : TIME;
	SettledBuffer : BOOL;
	O_OpenSP2BufferStop : BOOL;
	O_SelectPoint : BOOL;
	SP2BufferFull : BOOL;
	SP2BufferFullET : UDINT;
	ParingLoopEnabled : BOOL;
	BagInLoopHasDest : BOOL;
	O_OpenSDC1BufferStop : BOOL;
	BagSettledAtBuffer : BOOL;
	BagSettledAtBufferET : UDINT;
	Alternator : USINT;
	I_PaddleInPosition : BOOL;
	I_BagInIncline : BOOL;
	O_OpenBufferStop : BOOL;
	O_RunMotor : BOOL;
	I_BagAtOutgoingBuffer : BOOL;
	O_OutgoingBufferOpen : BOOL;
	BagSettled : BOOL;
	BagSettledET : UDINT;
	BagNearTop : BOOL;
	BagNearTopET : UDINT;
	CloseBufferStop : BOOL;
	CloseBufferStopET : UDINT;
	RunOn : BOOL;
	RunOnET : UDINT;
	I_BagOutAtTop : BOOL;
	BagAtBuffer : BOOL;
	BagAtBufferET : UDINT;
	I_BagStackerNearFull : BOOL;
	BagStackerHasSpace : BOOL;
	BagStackerHasSpaceET : UDINT;
	SIC3BufferFull : BOOL;
	SIC3BufferFullET : UDINT;
	HaltDownStairs : BOOL;
	SPL1BufferOpen : BOOL;
	SPITransitBag : BOOL;
END_VAR
```

#### 12_sp2Cyclic.ab
```automation-basic
PROGRAM _CYCLIC
	(* cyclic program *)

;---------------------------------------
;Sequence 12 - SP2 Single point 2 D[912]
;---------------------------------------

;Inputs

I_BagAtBuffer			= X[11].X15
I_PaddleInPosition		= X[10].X16
I_BagInIncline			= X[10].X15
I_BagOutAtTop           = X[11].X16
HaltDownStairs          = NOT X[6].X12

O_OpenBufferStop		= FALSE
O_RunMotor 				= FALSE

SPL1BufferOpen          = Y[9].Y01

I_BagAtOutgoingBuffer	= FALSE
O_OutgoingBufferOpen	= FALSE

Enable.IC[2]			= FALSE

Alarm[25].Name 			= 0
Alarm[25].Bag			= 284
Alarm[25].Beacon		= TRUE
Alarm[25].Extra			= 0
Alarm[25].Time			= 3000

;Setup Sequence
;STEP = D[925]
;Setup Pulse contact
PLS = (STEP <> LASTSTEP)
LASTSTEP = STEP

;Sequence
;Step 0 - Disabled
IF (STEP = 0) THEN
	;Disabled
ENDIF

;Run Incline until paddle in position
IF (STEP = 1) THEN
	O_RunMotor = NOT I_PaddleInPosition
	IF I_PaddleInPosition THEN
	;	D[925] = 2
	ENDIF
	IF NOT Std.EStop THEN
		Alarm[25].Name = almSwitchFault
	ENDIF
ENDIF

;Wait for at buffer
TON_10ms(I_BagAtBuffer AND (Bag[284].Cat > 0),300,BagAtBuffer,BagAtBufferET)
SPITransitBag = ((D[926] < 3) OR (D[926] > 5))
IF (STEP = 2) THEN
	IF (BagAtBuffer AND NOT SPL1BufferOpen AND SPITransitBag AND NOT HaltDownStairs) THEN
;		D[925] = 3
	ENDIF
	IF (Bag[284].Cat > 0) AND NOT I_BagAtBuffer THEN
		Alarm[25].Name 	= almBagNotAtProx
		Alarm[25].Bag	= 284
	ELSE IF (Bag[284].Cat = 0) AND I_BagAtBuffer THEN
		Alarm[25].Name 	= almBagNotShownOnScreen
		Alarm[25].Bag	= 284
	ENDIF
ENDIF

;Open Buffer stop
IF (STEP = 3) THEN
	O_OpenBufferStop 	= TRUE
	IF ((Bag[284].Cat > 0) AND (Bag[288].Cat = 0)) THEN
		Bag[288] = Bag[284]
		Bag[284] = Bag[0]
	ENDIF
	IF I_BagInIncline THEN
	;	D[925] = 4
	ENDIF
	Alarm[25].Name = almBagNotArrived
ENDIF

;Let bag settle at base of incline
TON_10ms((STEP = 4),700,BagSettled,BagSettledET)
IF (STEP = 4) THEN
	;O_OpenBufferStop 	= TRUE
	IF PLS THEN
		Bag[283] = Bag[288]
		Bag[288] = Bag[0]
	ENDIF
	IF BagSettled THEN
	;	D[925] = 5
	ENDIF
ENDIF

;Move Bag up incline
TON_10ms((STEP = 5),500,BagNearTop,BagNearTopET)
TON_10ms(((STEP = 5) AND NOT I_BagInIncline),1000,CloseBufferStop,CloseBufferStopET)
IF (STEP = 5) THEN
	;O_OpenBufferStop 	= NOT CloseBufferStop
	O_RunMotor 			= NOT BagNearTop
	IF BagNearTop THEN
	;	D[925] = 6
	ENDIF
	Alarm[25].Name = almSwitchFault
ENDIF

;Check for space at the ongoing buffer
;Run motor for 0.5 seconds
TON_10ms((STEP = 6),50,RunOn,RunOnET)
IF (STEP = 6) THEN
	O_RunMotor = NOT RunOn
	IF ((Bag[283].Cat > 0) AND (Bag[282].Cat = 0)) THEN
		Bag[282] = Bag[283]
		Bag[283] = Bag[0]
	ENDIF
	IF NOT Std.HaltSys THEN
		IF Line[18].Clear AND NOT I_BagOutAtTop AND (Bag[280].Cat = 0) THEN
	;		D[925] = 7
		ENDIF
	ENDIF
ENDIF

;Run incline until bag released / arrive at buffer
IF (STEP = 7) THEN
	O_RunMotor = TRUE
	IF PLS THEN
		C[18] = 0
	ENDIF
	IF Line[18].Trip THEN
		Bag[282].Dst = 0
		Bag[280]    = Bag[282]
		Bag[282]    = Bag[0]
	;	D[925] 		= 1
	ENDIF
	Alarm[25].Name = almBagNotReleased
ENDIF

;Alarms
TimerAlarm.IN 	= NOT PLS AND (Alarm[25].Name > 0)
TimerAlarm.PT 	= Alarm[25].Time
TimerAlarm FUB TON_10ms()
Alarm[25].On 	= TimerAlarm.Q
Alarm[25].ET 	= TimerAlarm.ET

;Outputs
;Y[11].Y15 = O_OpenBufferStop
;Y[13].Y07 = O_RunMotor
END_PROGRAM
```

### Program Logical/Sequences/10ms/26_spi1 (IEC, version 1.00.0) - * SPI1 Pneumatic Incline Up 1

#### 11_spi1Cyclic.ab
```automation-basic
PROGRAM _CYCLIC
	(* cyclic program *)

;Sequence 11 - Pneumatic Incline 1 D[911]

;Incline Conveyor

;-----------------------------------------
;Revision 1.00 17/01/2006 D.J. First Issue
;-----------------------------------------

I_BagAtBufferStop        = X[9].X02
I_CarriageAtTop          = X[9].X05
I_CarriageAtBottom       = X[9].X04
I_BagAtBottom            = X[9].X03
;I_BagReleased            = X[10].X14

SIC4BufferOpen          = Y[11].Y15
O_OpenBufferStop		= FALSE
O_SendCarriageDown      = FALSE

;Request.CPI[1]          = FALSE

;Setup Sequence
STEP = D[926]
;Setup Pulse contact
PLS = (STEP <> LASTSTEP)
LASTSTEP = STEP

Alarm[26].Name 			= 0
Alarm[26].Bag			= 10002
Alarm[26].Beacon		= TRUE
Alarm[26].Extra			= 0
Alarm[26].Time			= 3000

;Sequence
IF (STEP = 0) THEN
	;disabled
ENDIF

;wait for carriage at top
TON_10ms(I_CarriageAtTop,100,CarriageAtTop,CarriageAtTopET)
IF (STEP = 1) THEN

	IF CarriageAtTop  THEN
		D[926] = 2
	ENDIF
	Alarm[26].Name = almCarriageMoveFault
ENDIF

;request to CDC 1
IF ((STEP = 2) OR (STEP = 3)) THEN
	;Request.CPI[1] = TRUE
ENDIF

;check for bag at buffer
TON_10ms((I_BagAtBufferStop),200,BagAtBufferStop,BagAtBufferStopET)
IF (STEP = 2) THEN

	IF BagAtBufferStop AND NOT SIC4BufferOpen AND NOT Std.HaltSys THEN
			D[926] = 3
	ENDIF
	IF I_BagAtBottom OR I_CarriageAtBottom THEN
		Alarm[26].Name = almSwitchFault
	ENDIF
ENDIF

;Open buffer stop
IF (STEP = 3) THEN
		O_OpenBufferStop = TRUE

		IF I_BagAtBottom THEN
			D[926] = 4
		ENDIF
		Alarm[26].Name = almBagNotArrived
ENDIF

;wait for bag to settle
TON_10ms((I_BagAtBottom),200,BagAtBottom,BagAtBottomET)
IF (STEP = 4) THEN

		IF BagAtBottom THEN
			D[926] = 5
		ENDIF
		Alarm[26].Name = almBagNotSettled
ENDIF

;Send carriage down
TON_10ms((I_CarriageAtBottom),100,CarriageAtBottom,CarriageAtBottomET)
IF (STEP = 5) THEN
	O_SendCarriageDown = TRUE
	IF CarriageAtBottom THEN
		D[926] = 6
	ENDIF
	Alarm[26].Name = almCarriageMoveFault
ENDIF

;allow carriage to move up
IF (STEP = 6) THEN

	IF CarriageAtTop  THEN
		D[926] = 7
	ENDIF
	Alarm[26].Name = almCarriageMoveFault
ENDIF

;check buffer clear

IF (STEP = 7) THEN

	IF  Line[35].Clear AND BagAtBottom  THEN
		C[35]  = 0
		D[926] = 8
	ENDIF
	;Alarm[26].Name = almBagNotAtProx
ENDIF

;send carriage down
IF (STEP = 8) THEN
	O_SendCarriageDown = TRUE
	IF CarriageAtBottom THEN
		D[926] = 9
	ENDIF
	Alarm[26].Name = almCarriageMoveFault
ENDIF

;send carriage up
IF (STEP = 9) THEN
	IF CarriageAtTop  THEN
		D[926] = 1
	ENDIF
	Alarm[26].Name = almCarriageMoveFault
ENDIF

;wait for bag out
IF (STEP = 10) THEN
	IF Line[26].Trip THEN
		D[926] = 1
	ENDIF
	Alarm[26].Name = almBagNotArrived
ENDIF

;Alarms
TimerAlarm.IN 	= NOT PLS AND (Alarm[26].Name > 0)
TimerAlarm.PT 	= Alarm[26].Time
TimerAlarm FUB TON_10ms()
Alarm[26].On 	= TimerAlarm.Q
Alarm[26].ET 	= TimerAlarm.ET

;Outputs
;Y[10].Y12 = O_OpenBufferStop
Y[9].Y02 = O_SendCarriageDown
Y[9].Y01 = O_OpenBufferStop
END_PROGRAM
```

#### 11_spi1.var
```iecst
VAR RETAIN
	STEP : UINT;
	PLS : BOOL;
	LASTSTEP : UINT;
	BagSettled : BOOL;
	BagSettledET : TIME;
	O_OpenBufferStop : BOOL;
	BagSettledBuffer : BOOL;
	I_BaginIncline : BOOL;
	BagSettledBufferET : TIME;
	I_BagAtBuffer : BOOL;
	I_CarrAtBottom : BOOL;
	I_CarrAtTop : BOOL;
	O_MoveDown : BOOL;
END_VAR
VAR
	TempDownTime : BOOL;
	TempDownTimeET : TIME;
	I_BagAtBufferStop : BOOL;
	I_CarriageAtTop : BOOL;
	I_CarriageAtBottom : BOOL;
	I_BagAtBottom : BOOL;
	SIC4BufferOpen : BOOL;
	O_SendCarriageDown : BOOL;
	CarriageAtTop : BOOL;
	CarriageAtTopET : UDINT;
	BagAtBufferStop : BOOL;
	BagAtBufferStopET : UDINT;
	BagAtBottom : BOOL;
	BagAtBottomET : UDINT;
	CarriageAtBottom : BOOL;
	CarriageAtBottomET : UDINT;
	TimerAlarm : TON_10ms;
END_VAR
```

### Program Logical/Sequences/10ms/32_stb2 (IEC) - *For Reference only-- Adjust as required.

#### belt.var
```iecst
VAR
	myPrg : USINT;
	BeltAddTimeArray : ARRAY[0..59] OF UINT;
	mySeq : UINT;
	myOtherBeltSeq : UINT;
	myLuBag : UINT;
	myVCBag : UINT;
	PurgeBagIndex : UINT;
	Bank : UINT;
	myBelt : UINT;
END_VAR
VAR RETAIN
	MinBeltRunCV : UINT;
END_VAR
VAR
	STEP : UINT;
	n : UINT;
	myZone : UINT;
	myWgt : UINT;
	StnBag : UINT;
	LASTSTEP : UINT;
	PurgeReverseBagIndex : UINT;
	myOutBag : UINT;
	myOppBeltBag : UINT;
	BeltAddTime : UINT;
	BeltRunTime : UINT;
	VCBag : UINT;
	myBank : UINT;
	myBag : UINT;
	TrackingOkET : UDINT;
	myCus : UDINT;
	LinenDetectedRevET : UDINT;
	myCat : UDINT;
	BeltClearReverseET : UDINT;
	LinenDetectedReverseET : UDINT;
	BeltOKET : UDINT;
	TimerAlarm : TON_10ms;
	LinenIsDetectedET : TIME;
	LargeLoadClearET : TIME;
	Step6ET : TIME;
	LinenDetectedET : TIME;
	BeltClearET : TIME;
	MinimumRunET : TIME;
	myOppositeBelt : INT;
	CountValue : INT;
	WeightValue : INT;
	b : INT;
	MixCust : BOOL;
	BeltOK : BOOL;
	O_Reverse : BOOL;
	Purge : BOOL;
	LinenIsDetected : BOOL;
	MinimumRun : BOOL;
	PhotocellsClear : BOOL;
	MinBeltRunET : BOOL;
	O_SlowBelt : BOOL;
	LinenDetectedReverse : BOOL;
	BeltRunning : BOOL;
	PurgeReverse : BOOL;
	Stb2_Running : BOOL;
	LargeLoadClear : BOOL;
	I_PhotoLarge : BOOL;
	BeltClearReverse : BOOL;
	I_LinenAtEndSTB3 : BOOL;
	RunBelt : BOOL;
	I_PhotoBottom : BOOL;
	O_RunBelt : BOOL;
	LinenDetected : BOOL;
	StationOpen : BOOL;
	I_PhotoTop : BOOL;
	PLS : BOOL;
	MinBeltRun : BOOL;
	WeightValid : BOOL;
	I_DisableLoadingUnit : BOOL;
	LinenDetectedRev : BOOL;
	RunSlow : BOOL;
	I_PhotoReverse : BOOL;
	CountValid : BOOL;
	BeltClear : BOOL;
	TrackingOk : BOOL;
	myOtherBeltRunning : BOOL;
	myStnReg : UINT;
	myStnBit : UINT;
	myTimeStamp : DATE_AND_TIME;
	myHttp : UINT;
	catString : STRING[15];
	cusString : STRING[15];
	wgtString : STRING[15];
	batchString : STRING[32];
	requestURL : STRING[254];
	responseData : ARRAY[0..49] OF USINT;
	commaPos : INT;
	I_InvStatus : BOOL;
	myBagNumber : UINT;
	MixCats : BOOL;
	MixCusts : BOOL;
	MixProgs : BOOL;
	stnNo : USINT;
	I_Manual_Stop : BOOL;
END_VAR
```

#### _setBeltTime.st
```iecst
ACTION _setBeltTime:

BeltAddTimeArray[1] := 1;
BeltAddTimeArray[2] := 1;
BeltAddTimeArray[3] := 2;
BeltAddTimeArray[4] := 2;
BeltAddTimeArray[5] := 3;
BeltAddTimeArray[6] := 3;
BeltAddTimeArray[7] := 4;
BeltAddTimeArray[8] := 4;
BeltAddTimeArray[9] := 5;
BeltAddTimeArray[10] := 5;
BeltAddTimeArray[11] := 6;
BeltAddTimeArray[12] := 6;
BeltAddTimeArray[13] := 7;
BeltAddTimeArray[14] := 7;
BeltAddTimeArray[15] := 8;
BeltAddTimeArray[16] := 8;

END_ACTION
```

#### beltCyclic.ab
```automation-basic
PROGRAM _INIT
	_setBeltTime

END_PROGRAM

PROGRAM _CYCLIC
 	(* cyclic program *)

;Sequence 2 - Transfer Belt 1 from Stations 1-8

;-----------------------------------------
;Revision 1.00 18/01/2006 D.J. First Issue
;-----------------------------------------

;Inputs and Outputs
;-----------------

myBank 			= 2
myBelt			= 2
mySeq			= 33
myBag			= 162
myOutBag		= 160
myZone			= 0

MixCats			= (D[369] > 0)
MixCusts		= (D[366] > 0)	;Allow mixing of customers?
MixProgs		= (D[367] > 0)	;Allow mixing of Programs?

;I_PhotoBottom		      	= X[3].X08
I_PhotoTop   		      	= X[3].X02
I_Manual_Stop               = X[15].X04
I_PhotoReverse            	= FALSE
I_InvStatus					= TRUE

;Belt add times in an array for each station as station number will not work..
;LOOP n = 20 DOWNTO 1 DO
;	BeltAddTimeArray[n]		= n
;ENDLOOP

RequestRel.TransferBelt[myBelt]		  	= FALSE
Request.TransferBelt[myBelt]		    = FALSE

O_RunBelt 					= FALSE
O_Reverse					= FALSE
O_SlowBelt					= FALSE

;Check all stations are closed.
StationOpen = FALSE
LOOP n = 1 TO Ldg[myBank].NoStations DO
	stnNo = Ldg[myBank].Stations[n]
	IF (D[950 + stnNo] = 3) THEN
		StationOpen = TRUE
	ENDIF
ENDLOOP

Alarm[mySeq].Name 				= 0
Alarm[mySeq].Bag				= myBag
Alarm[mySeq].Beacon				= FALSE
Alarm[mySeq].Extra				= 0
Alarm[mySeq].Time			  	= 5000

;n = D[900 + Std.StationBankReg + myBank] ;Selected Station
n = D[900 + 50]

STEP = D[900 + mySeq]
;Setup Pulse contact
PLS = (STEP <> LASTSTEP)
LASTSTEP = STEP

;Step 0 - Disabled
IF STEP = 0 THEN
	;Disabled
ENDIF

;Step 1 - Check no stations are releasing
IF STEP = 1 THEN
	;Don't allow stations to release
	Ldg[myBank].EnableStnRelease = FALSE
	Std.PurgeBank[myBank].PurgeOn = 0 ; Clear to display Purge
	Std.PurgeBank[myBank].StationsStatus[0] = 0 ;trackview TO display Purge
	Std.PurgeBank[myBank].StationsStatus[1] = 0
	;No Station Releaseng and switched on
	IF (NOT StationOpen AND (D[mySeq] > 0) AND NOT I_Manual_Stop) THEN
		IF (Bag[myBag].Cat = 0) THEN
			D[900 + mySeq] = 2 ;No Bag on belt
		ELSE
			D[900 + mySeq] = 4 ;Bag on belt
		ENDIF
	ENDIF
	Alarm[mySeq].Name = almNoAlarm
ENDIF

;Step 2 - Enable Station search
IF STEP = 2 THEN
	IF (Bag[myBag].Cat > 0) THEN
;		D[900 + mySeq] = 4
	ENDIF
	;Check each station to see if a manual destination has been set
	LOOP n = 1 to Ldg[myBank].NoStations DO

		//StnBag = Std.StationBagsStart + Ldg[myBank].Stations[n] - 1
		StnBag = LDG_GetBagFromStation(Std.StationBagsStart,n)

		IF ((Bag[StnBag].Dst > 0) AND (Bag[StnBag].Dst < 99) AND (D[mySeq] > 0)) THEN ;Dest 99 = Empty Bag in station
			Stn[n].DestManual = Bag[StnBag].Dst
		ELSE
			Stn[n].DestManual = 0
		ENDIF
		;For pairing set number of spaces to search for
		Stn[n].SpacesRequired = 1 ;D[2000 + Bag[StnBag].Prg]

	ENDLOOP

	;Station Search

	IF ((Ldg[myBank].Search = 0) AND (D[mySeq] > 0) AND NOT Std.HaltSysZone[myZone] AND EnableRel.TransferBelt[myBelt])  THEN
		Ldg[myBank].Search = 1
		PurgeBagIndex = 0
	ELSE IF ((Ldg[myBank].Search = 2) AND (Ldg[myBank].Found > 0)) THEN ;
		IF (Ldg[myBank].Found < 97) THEN
			D[900 + 50] 	= Ldg[myBank].Found
			n 	= D[900 + 50]
;		ELSE IF (Ldg[myBank].Found = 98) OR (Ldg[myBank].Found = 97) THEN ; Reverse belt
;			D[900 + mySeq] = 9
;			GOTO ExitStep2 ; Ignore the rest of Step 2
		ELSE
;			IF (Ldg[myBank].Found = 98) OR (Ldg[myBank].Found = 97) THEN
;				Ldg[myBank].Line = 21 ; Set Destination to SDC1
;			ENDIF
		;	Purge = TRUE

			n = LDG_GetStationFromBag(Std.StationBagsStart,Std.PurgeBank[myBank].PurgeBatch[PurgeBagIndex])
			IF (n = 0) OR (n > Ldg[myBank].Stations[Ldg[myBank].NoStations]) THEN
				Ldg[myBank].Search = 0
				GOTO ExitStep2
			ENDIF
			D[900 + 50] = n
			Std.PurgeBank[myBank].PurgeOn = 1 ; Send to trackview to display Purge
			myStnReg = (n > 32)
			IF (myStnReg = 0)THEN
				myStnBit =	n - 1
			ELSE IF (myStnReg = 1)THEN
				myStnBit = 	n - 33
				ELSE
				myStnBit = 0
			ENDIF
			Std.PurgeBank[myBank].StationsStatus[myStnReg] = BIT_SET(Std.PurgeBank[myBank].StationsStatus[myStnReg],myStnBit)
			;Get highest belt add time... Use array as station numbers are opposite to distanct
			IF BeltAddTimeArray[n] > BeltAddTime THEN
				BeltAddTime = BeltAddTimeArray[n]
			ENDIF
		ENDIF
		StnBag = LDG_GetBagFromStation(Std.StationBagsStart,n)
		;Clear the release button count if used
		Stn[n].ManualRelease 	= FALSE
		Stn[n].Purge 			= FALSE
		Stn[n].PurgeReverse	 	= FALSE
		Stn[n].PBCount 			= 0
		;------Write Report------
	;	IF Std.StationReports AND (Ldg[myBank].Found <> 98) AND (Ldg[myBank].Found <> 97)THEN
        IF Std.StationReports THEN
			IF (ReportLoading[n].Cat = 0)  THEN
				IF Purge THEN
					IF (PurgeBagIndex < Std.PurgeBank[myBank].PurgeBagQty) THEN
						PurgeBagIndex = PurgeBagIndex + 1
					ENDIF
				ENDIF
				WeightValue = Stn[n].Weight - INT(StnPrev[n].Wgt)
				WeightValid = (WeightValue > 0)

				;Check if anything has been added and current weight is not less than the previous
				CountValue = Stn[n].Count - INT(StnPrev[n].Cnt)
				CountValid = (CountValue > 0)
				IF (WeightValid OR CountValid) THEN
					;Ensure valid values as we report on either a weight or count change
					IF (WeightValue < 0) THEN
						WeightValue = 0
					ENDIF

					IF (CountValue < 0) THEN
						CountValue = 0
					ENDIF
					myTimeStamp = CurrentTimestamp
					ReportLoading[n].Prg = Bag[StnBag].Prg 			;Program
					ReportLoading[n].Cat = Bag[StnBag].Cat			;Category
					ReportLoading[n].Cus = Bag[StnBag].Cus			;Customer
					ReportLoading[n].Wgt = UINT(WeightValue)		;Weight
					ReportLoading[n].Cnt = UINT(CountValue)			;Count
					ReportLoading[n].Stn = n         				;Station
					ReportLoading[n].Mcn = 0						;Machine
					ReportLoading[n].Bid = Bag[StnBag].Bid			;Batch ID
					ReportLoading[n].TimeStamp = myTimeStamp

				ENDIF
			ENDIF
		ELSE
			myTimeStamp = CurrentTimestamp
			IF Purge THEN
				IF (PurgeBagIndex < Std.PurgeBank[myBank].PurgeBagQty) THEN
					PurgeBagIndex = PurgeBagIndex + 1
				ENDIF
			ENDIF
		ENDIF

		;Set Previous Cat and Cus to Current and Clear Weight and Count
		StnPrev[n].Prg 	= Bag[StnBag].Prg
		StnPrev[n].Cat 	= Bag[StnBag].Cat
		StnPrev[n].Cus 	= Bag[StnBag].Cus
		StnPrev[n].Wgt 	= 0
		StnPrev[n].Cnt 	= 0
		StnPrev[n].Bid 	= Bag[StnBag].Bid

		Ldg[myBank].EnableStnRelease = TRUE
		;Clear Manual Release and Count
		Stn[n].ManualRelease 	= FALSE
		Stn[n].Count			= 0
		BeltAddTime = BeltAddTimeArray[n]
		;Keep A record of purged bags to attach the data for the biggest loads
		IF Purge THEN
			//Set the category Number
			IF Ldg[Bank].Found = 97 THEN // 97 is weight too small so always set to mixed so it doesn;t get sent to washer..
				myCat = CAT_MIXED_LINEN //Std.MaxCats	- 1
				myPrg = Std.MaxProg	- 1
			ELSE IF (myCat > 0) AND (Bag[StnBag].Cat <> myCat) THEN
				IF (MixCats OR MixProgs) THEN
					//Take the Cat code of bag with most weight
					IF (Bag[StnBag].Wgt > myWgt) THEN
						myCat = Bag[StnBag].Cat
						myPrg = Bag[StnBag].Prg
						myWgt = Bag[StnBag].Wgt
					ENDIF
				ELSE //Different Cats in 1 bag
					myCat = CAT_MIXED_LINEN//Std.MaxCats	- 1
					myPrg = Std.MaxProg - 1
				ENDIF
			ELSE
				myCat = Bag[StnBag].Cat
				myPrg = Bag[StnBag].Prg
				myWgt = Bag[StnBag].Wgt
			ENDIF

			IF (myCus > 0) AND (Bag[StnBag].Cus <> myCus) THEN
				myCus = Std.MaxCust - 1
			ELSE
				myCus = Bag[StnBag].Cus
			ENDIF
		ENDIF

		IF Purge AND (PurgeBagIndex = Std.PurgeBank[myBank].PurgeBagQty) THEN ;Do not minus 1 from purge qty as the indexing is above so will always read 1 more..
			Bag[myBag] 		= Bag[StnBag]
			Bag[StnBag].Mis = 0
			Bag[StnBag].Bid = 0 ; Reset BID

			Bag[myBag].Cat = myCat
			Bag[myBag].Prg = myPrg
			Bag[myBag].Ur2 = 99
			Bag[myBag].Cus	= myCus
			Bag[myBag].Dst 	= USINT(Ldg[myBank].Line)	;Destination
			Bag[myBag].Wgt 	= Std.PurgeBank[myBank].PurgeBatchWieght
			Bag[myBag].Cnt 	= Std.PurgeBank[myBank].PurgeBatchCount

			Bag[myBag].Timestamp = myTimeStamp
			Bag[StnBag].Bid = 0 ; Reset BID
			Bag[StnBag].Dst = 0 					;Reset Destination (Manual)
			Bag[StnBag].Mis = 0
			IF (Ldg[myBank].Found = 98) OR (Ldg[myBank].Found = 97) THEN
	;			D[900 + mySeq] = 3 ;Reverse belt not used.
			ELSE
	;			D[900 + mySeq] = 3
			ENDIF
		ELSE IF NOT Purge AND (Bag[StnBag].Cat <> 98) THEN
			;Copy Station Data to Belt Bag
			Bag[myBag] 		= Bag[StnBag]
			Bag[myBag].Dst 	= USINT(Ldg[myBank].Line)	;Destination
			Bag[myBag].Ur2 = StnBag
			Bag[StnBag].Bid = 0 ; Reset BID
			Bag[StnBag].Dst = 0; USINT(Ldg[myBank].Line) 					;Reset Destination (Manual)
			Bag[StnBag].Mis = 0
			Bag[myBag].Timestamp = myTimeStamp
        	D[900 + mySeq] = 3
		ENDIF
		Alarm[mySeq].Name = almNoAlarm
	ENDIF
ELSE
	Purge = FALSE
	PurgeBagIndex		= 0
	Ldg[myBank].Search  	= 0 ;Clear Search if not on step 2
	myCat = 0
	myPrg = 0
	myCus = 0
	myWgt = 0
ENDIF
ExitStep2:

;;Get batch ID from SQL Server
;IF ((STEP >= 3) AND (STEP <= 4)) THEN
;	IF (Bag[myBag].Mis = 0) THEN
;		_httpRequest;
;	ENDIF
;ELSE
;	HTTP_Comm[myHttp].Status = HTTP_COMM_STATUS_DISABLED
;ENDIF

;Step 3
;Release to Belt Conveyor
TON_10ms(I_PhotoTop,10,LinenDetected,LinenDetectedET)
IF (STEP = 3) THEN
	O_RunBelt = TRUE
	IF LinenDetected OR Test.TransferBelt THEN
		D[900 + mySeq] = 4
	ENDIF
	Alarm[mySeq].Name = almPhotocellNotMade
ENDIF

TON_10ms((STEP = 4),10,RunBelt,Step6ET)
IF (STEP = 4) THEN

	RequestRel.TransferBelt[myBelt] = (Bag[myBag].Cat > 0)
	n = D[900 + 50]
	IF EnableRel.TransferBelt[myBelt]  THEN; AND (Bag[myBag].Mis > 0)
		;myTimeStamp = CurrentTimestamp
;		ReportLoading[n].Prg = Bag[290].Prg 			;Program
;		ReportLoading[n].Cat = Bag[290].Cat			;Category
;		ReportLoading[n].Cus = Bag[290].Cus			;Customer
;		ReportLoading[n].Wgt = UINT(WeightValue)		;Weight
;		ReportLoading[n].Cnt = UINT(CountValue)			;Count
;		ReportLoading[n].Stn = n         				;Station
;		ReportLoading[n].Mcn = 0						;Machine
;		ReportLoading[n].Bid = Bag[290].Bid			;Batch ID
;		ReportLoading[n].Mis = Bag[290].Mis
;		ReportLoading[n].TimeStamp = Bag[290].Timestamp
		D[900 + mySeq] = 5
	ENDIF
	IF (Bag[myBag].Cat = 0) THEN
		Alarm[mySeq].Name = almBagDataError
	ELSE IF (Bag[myBag].Mis = 0) THEN
	;	Alarm[mySeq].Name = almBagDataError
	ENDIF

ENDIF

;Step 5 - Run Belt until linen detected for 1 second and Station has emptied
TON_10ms(((STEP = 5) AND I_PhotoTop AND I_InvStatus),50,LinenIsDetected,LinenIsDetectedET)
IF (STEP = 5) THEN
	O_RunBelt = TRUE
	Ldg[myBank].EnableStnRelease = TRUE ;Enable Station to Open bags if they haven't been already
	IF (LinenIsDetected OR Test.TransferBelt)   THEN
		D[900 + mySeq] = 6
	ENDIF
	IF (Bag[myBag].Cat = 0) OR (Bag[myOutBag].Cat > 0) THEN
		Alarm[mySeq].Name = almBagDataError
	ELSE IF NOT Std.HaltSysZone[myZone] THEN
		Alarm[mySeq].Name = almPhotocellNotMade
	ENDIF
ENDIF

;Step 6 - Run Belt until photocells clear for 12 seconds
;TON_10ms((STEP = 6),200,MinimumRun,MinimumRunET)
TON_10ms(((STEP = 6) AND I_InvStatus  AND NOT I_PhotoTop AND NOT Std.HaltSysZone[myZone]),500,BeltClear,BeltClearET)
IF (STEP = 6) THEN
	O_RunBelt = TRUE
	IF (BeltClear AND MinBeltRun AND (Bag[myBag].Cat > 0) AND ((Bag[myOutBag].Cat = 0) OR (Bag[myOutBag].Cat = Std.MaxCats))) THEN
		myBagNumber = Bag[myOutBag].Ur1
		Bag[myOutBag] = Bag[myBag]
		Bag[myOutBag].Ur1 = myBagNumber
		Bag[myBag] = Bag[0]
		D[900 + mySeq] = 7
	ENDIF
	IF NOT Std.HaltSysZone[myZone] THEN
		IF I_PhotoBottom OR I_PhotoTop THEN
			Alarm[mySeq].Name = almPhotocellBlocked
		ELSE IF StationOpen THEN
			Alarm[mySeq].Name = almStationNotClosed
		ELSE IF NOT MinBeltRun THEN
			Alarm[mySeq].Name = almClearingBeltPleaseWait
		ENDIF
	ENDIF
ENDIF

;Step  - Check Stations Are Closed
IF (STEP = 7) THEN
	IF NOT StationOpen AND (Bag[myBag].Cat = 0) THEN
		D[900 + mySeq] = 1
	ENDIF
	Alarm[mySeq].Name = almStationNotClosed
ENDIF

;Note - Unitl the Station has closed the min belt run time won't start
BeltRunTime = (12 + BeltAddTime)
;CTU((O_RunBelt AND Std.Clock1s AND (D[900 + Std.StationBankReg + myBank] = 0) AND NOT Std.EStop),(STEP = 1),BeltRunTime,MinBeltRun,MinBeltRunCV)
BeltRunning = (O_RunBelt OR O_Reverse)
CTU((BeltRunning AND I_InvStatus AND Std.Clock1s AND NOT StationOpen  AND NOT Std.HaltSysZone[myZone]),(STEP = 1),BeltRunTime,MinBeltRun,MinBeltRunCV)

;Slow speed for large load on belt
TON_10ms((NOT I_PhotoLarge AND NOT RunSlow),300,LargeLoadClear,LargeLoadClearET)
IF ((STEP > 2) AND (STEP < 7)) THEN
	IF I_PhotoLarge THEN
		O_SlowBelt = TRUE
	ENDIF
ENDIF

IF (STEP > 0) AND NOT I_InvStatus	THEN
	Alarm[mySeq].Name = almMotorOverload
	Alarm[mySeq].Time = 0
ENDIF

;Alarms
TimerAlarm.IN = NOT PLS AND (Alarm[mySeq].Name > 0)
TimerAlarm.PT = Alarm[mySeq].Time
TimerAlarm FUB TON_10ms()
Alarm[mySeq].On = TimerAlarm.Q
Alarm[mySeq].ET = TimerAlarm.ET

;Outputs
;Inform Station Sequences that the belt has been
Ldg[myBank].BeltHasRun =  (((((D[900 + mySeq] > 3) AND (D[900 + mySeq] < 7)) OR (D[900 + mySeq] >= 10)) AND Ldg[myBank].EnableStnRelease)  OR (D[900 + mySeq] = 1))

Y[11].Y13 = O_RunBelt
//Y[8].Y03 = O_RunBelt AND (STEP < 7) ; Inclined belt... Do not run when reversing.
//Y[8].Y02 = O_Reverse

END_PROGRAM
```

### Program Logical/Sequences/10ms/44_pn (IEC) - *Ongoing Sequence

#### x_pn.var
```iecst
VAR
	AlarmOld : UINT;
	Area : UINT;
	AreaChoice : ARRAY[0..4] OF UINT;
	AreaEndLine : UINT;
	AreaStartLine : UINT;
	AreaValid : BOOL;
END_VAR
VAR RETAIN
	Buff : UINT;
END_VAR
VAR
	Buffer : UINT;
	BufferBag : UINT;
	BufferBagNum : ARRAY[0..4] OF UINT;
	BufferCat : UDINT;
	BufferCus : UDINT;
	BufferDst : UINT;
	BufferPrg : UINT;
	BufferSettled : BOOL;
END_VAR
VAR RETAIN
	Dest : UINT;
END_VAR
VAR
	FoundDepth : UINT;
	I_BagatBuffer : ARRAY[0..4] OF BOOL;
END_VAR
VAR RETAIN
	LASTSTEP : UINT;
	LineSelect : ARRAY[0..19] OF BOOL;
END_VAR
VAR
	MaxBuffers : UINT;
	MaxDepth : UINT;
	MaxLine : UINT;
	MinLine : UINT;
	myDepth : UINT;
	myFound : UINT;
	myLine : UINT;
	myLineUsed : BOOL;
	myLineValid : BOOL;
	mySpace : UINT;
	n : UINT;
	O_OpenSelect : ARRAY[0..4] OF BOOL;
	O_Reset : BOOL;
	OnGoingEnable : BOOL;
END_VAR
VAR RETAIN
	PLS : BOOL;
END_VAR
VAR
	ResetPoints : BOOL;
	ResetPointsET : TIME;
	SearchBag : UINT;
	SettledBuffer : ARRAY[0..4] OF BOOL;
	SettledBufferET : ARRAY[0..4] OF TIME;
END_VAR
VAR RETAIN
	STEP : UINT;
END_VAR
VAR
	TestBuffer : UINT;
	TimerAlarm : TON_10ms;
	I_BagBagReleased : BOOL;
	mySeq : UINT;
	myZone : UINT;
	myTransitBag : UINT;
	myStartStop : UINT;
	O_OpenBuffer : ARRAY[0..9] OF BOOL;
	PairLoopSpace : BOOL;
	Bfr : INT;
	DestValid : BOOL;
END_VAR
```

#### x_pn.ab
```automation-basic
PROGRAM _CYCLIC

;--------------------------------------
;Sequence 4 - Ongoing To Storage D[900 + mySeq]
;--------------------------------------

;--------------------------------------------------------------------------------
;Revision 1.00 06/11/2009 D.J. First Issue - Automatic Line Allocation with Areas
;--------------------------------------------------------------------------------
OnGoingEnable 		= ((D[14] > 0) AND NOT Std.HaltSys)

I_BagatBuffer[1]	= FALSE
I_BagatBuffer[2]	= FALSE ;X[7].X14
I_BagatBuffer[3]	= FALSE
I_BagatBuffer[4]	= FALSE

O_Reset 		  	= FALSE
O_OpenSelect[1]		= FALSE
O_OpenSelect[2]		= FALSE
O_OpenSelect[3]		= FALSE
O_OpenSelect[4]		= FALSE

Enable.SVC3HighLevel= FALSE
Enable.SVC2AtTop    = FALSE
Request.SP[2] 		= FALSE

Alarm[4].Name 		= 0
Alarm[4].Bag		= 151
Alarm[4].Beacon		= TRUE
Alarm[4].Extra	 	= 0
Alarm[4].Time		= 3000

;Setup Sequence
;--------------
STEP = D[904]
;Setup Pulse contact
PLS = (STEP <> LASTSTEP)
LASTSTEP = STEP

;Check if Recirculation bag needs a destination
;IF ((Bag[107].Cat > 0) AND (Bag[107].Dst = 0) AND (D[1005] > 0) AND (D[1005] <= 6) AND (D[1006] > 0)) THEN
;	Bag[107].Dst 	= D[1005]
;	D[1006] 		= (D[1006] - 1)
;ENDIF

;Step 0 - Disabled
IF (STEP = 0) THEN
	;Disabled
ENDIF

;Step 1 - Reset Ongoing Points
TON_10ms((STEP = 1),300,ResetPoints,ResetPointsET)
IF (STEP = 1) THEN
	Dest  	= 0
	Buff 	= 0
	O_Reset = TRUE
	IF (ResetPoints AND OnGoingEnable) THEN
		D[904] = 2
	ENDIF
ENDIF

;Set Max Buffers to search
MaxBuffers = 2

;Bag Settles at each buffer
TON_10ms(Request.SVC2AtTop,100,SettledBuffer[1],SettledBufferET[1]) ;sequence 9 on step 8 and no PairedBag on loop
TON_10ms(Request.SVC3HighLevel,100,SettledBuffer[2],SettledBufferET[2]);sequence 10 on step 7

BufferBagNum[1]	= 296 ;svc 2 bag
BufferBagNum[2]	= 310 ;svc 3 bag

;Step 2 - Search for a valid Bag at one of the buffers
Line[12].Space = PairLoopSpace
IF (STEP = 2) THEN

	Buff 	= 0
	Dest 	= 0

	IF OnGoingEnable THEN

		Alarm[4].Name 	= almNoAlarm
		Alarm[4].Time	= 2000

		LOOP Bfr = 1 TO MaxBuffers DO

			;Set Test Value for Monitoring
			IF TestBuffer > 0 THEN
				Buffer = TestBuffer
			ELSE
				Buffer = Bfr
			ENDIF

			BufferBag		= BufferBagNum[Buffer]
			BufferSettled 	= SettledBuffer[Buffer]
			BufferCat 		= Bag[BufferBag].Cat
			BufferDst 		= Bag[BufferBag].Dst

			DestValid = ((BufferDst >= 6) AND (BufferDst <= 12))

			IF (BufferSettled AND (BufferCat > 0) AND DestValid AND (Bag[298].Cat = 0)) THEN
				n = BufferDst

				IF ((n >= 6) AND (n <= 11) AND (Line[n].Space > 0) AND Line[n].Clear) THEN
					Dest 	= n
					Buff 	= Buffer
					D[904] 	= 3
				ELSE IF (n = 12) THEN
					Request.SP[2] = TRUE
					IF Enable.SP[2] THEN
						Dest 	= n
						Buff 	= Buffer
						D[904]  = 3
					ENDIF
				ELSE
					Alarm[4].Name 	= almDestinationNotValid
					Alarm[4].Bag	= BufferBag
				ENDIF
			ENDIF

			;Buffer Alarms
			;IF (BufferCat > 0) AND NOT BufferSettled THEN
			;	Alarm[4].Name 	= almBagNotAtProx
			;	Alarm[4].Bag	= BufferBag
			;ELSE IF (BufferCat = 0) AND BufferSettled THEN
			;	Alarm[4].Name 	= almBagNotShownOnScreen
			;	Alarm[4].Bag	= BufferBag
			;ENDIF

		ENDLOOP

	ENDIF

ENDIF

;Clear Line Selections
LOOP n = 6 TO Std.MaxLines DO
	LineSelect[n] = FALSE
ENDLOOP

;Step 3 - Enable SVC2 or SVC3 to Release a bag
IF (STEP = 3) THEN

	LineSelect[Dest] 		= TRUE
	Request.SP[2]			= (Dest = 12)

	Enable.SVC2AtTop 		= (Buff = 1)
	Enable.SVC3HighLevel 	= (Buff = 2)

	IF PLS THEN
		C[Dest] = 0
		IF (Bag[298].Cat = 0) AND (Bag[BufferBagNum[Buff]].Cat > 0) THEN
			Bag[298]				 	= Bag[BufferBagNum[Buff]]
			Bag[BufferBagNum[Buff]]	 	= Bag[0]
		ENDIF
	ENDIF

	;Bag released from SVC2
	IF ((Buff = 1) AND NOT Request.SVC2AtTop) THEN
		D[904] = 4
	ENDIF

	;Bag released from SVC3
	IF ((Buff = 2) AND NOT Request.SVC3HighLevel) THEN
		D[904] = 4
	ENDIF

ENDIF

;Step 4 - Select line / open buffer stop
IF (STEP = 4) THEN

	LineSelect[Dest] 		= TRUE
	Request.SP[2]			= (Dest = 12)

	;Bag arrived on selected line
	IF Line[Dest].Trip THEN
		D32[498] 						= Bag[298].Cus	;Set Customer for Customer FIFO
		Bag[298].Dst 				= 0 		    ;Clear Destination
		Bag[Line[Dest].LastBag] 	= Bag[298]
		Bag[298] 					= Bag[0]
		D[904] 						= 1
	ENDIF

	Alarm[4].Name = almBagNotArrived

ENDIF

;Alarms
TimerAlarm.IN = NOT PLS AND (Alarm[4].Name > 0) AND (AlarmOld = Alarm[4].Name)
TimerAlarm.PT = Alarm[4].Time
TimerAlarm FUB TON_10ms()
Alarm[4].On = TimerAlarm.Q
Alarm[4].ET = TimerAlarm.ET

AlarmOld = Alarm[4].Name ;Need to ensure alarm changes as may be multiple alarms on step 2

;Outputs
Y[4].Y06 = LineSelect[6]
Y[4].Y07 = LineSelect[7]
Y[4].Y08 = LineSelect[8]
Y[4].Y09 = LineSelect[9]
Y[4].Y10 = LineSelect[10]
Y[4].Y11 = LineSelect[11]
Y[4].Y15 =  O_Reset

END_PROGRAM
```

### Program Logical/Sequences/10ms/23_spr3 (IEC, version 1.00.2) - *Pressure Relief
